# B&R Automation Studio project Panasonic_LinkaPowerCP2_A2021055 (part 27)

#### AtlasCopcoKomunikacia.st
```iecst
ACTION AtlasCopcoKomunikacia:

    M5_PrevodMomentu();
    K40_PrevodMomentu();

	//**************************************************************Skrutkovacka M5**************************************************************//
	//Vstupy z AtlasCopco do PLC//
    P3_Srobovanie.Skrutkovacka_M5.Stav_VysledokPotvrdeny:= P3_Srobovanie.PAR.M5_AtlasCopcoInputs[0].0;
    P3_Srobovanie.Skrutkovacka_M5.Stav_EmergencyStop:= P3_Srobovanie.PAR.M5_AtlasCopcoInputs[0].1;
    P3_Srobovanie.Skrutkovacka_M5.Stav_READY_to_START:= P3_Srobovanie.PAR.M5_AtlasCopcoInputs[0].2;
    P3_Srobovanie.Skrutkovacka_M5.Stav_MANUAL:= P3_Srobovanie.PAR.M5_AtlasCopcoInputs[0].3;
    P3_Srobovanie.Skrutkovacka_M5.Stav_UtahovanieUkoncene:= P3_Srobovanie.PAR.M5_AtlasCopcoInputs[0].4;
    P3_Srobovanie.Skrutkovacka_M5.Stav_VysledokUtahovania_NG:= P3_Srobovanie.PAR.M5_AtlasCopcoInputs[0].5;
    P3_Srobovanie.Skrutkovacka_M5.Stav_VysledokUtahovania_OK:= P3_Srobovanie.PAR.M5_AtlasCopcoInputs[0].6;
    P3_Srobovanie.Skrutkovacka_M5.Stav_SmerOtacania_VPRED:= P3_Srobovanie.PAR.M5_AtlasCopcoInputs[0].7;
    P3_Srobovanie.Skrutkovacka_M5.Stav_BUSY:= P3_Srobovanie.PAR.M5_AtlasCopcoInputs[0].8;
    P3_Srobovanie.Skrutkovacka_M5.Stav_ControlerSwitch_ON:= P3_Srobovanie.PAR.M5_AtlasCopcoInputs[0].9;
    P3_Srobovanie.Skrutkovacka_M5.Stav_Station_READY:= P3_Srobovanie.PAR.M5_AtlasCopcoInputs[0].10;
    P3_Srobovanie.Skrutkovacka_M5.Stav_NastrojPripojeny:= P3_Srobovanie.PAR.M5_AtlasCopcoInputs[0].11;
    P3_Srobovanie.Skrutkovacka_M5.Stav_NastrojUtahuje:= P3_Srobovanie.PAR.M5_AtlasCopcoInputs[0].12;

    //Výstupy z PLC do AtlasCopco//
    P3_Srobovanie.PAR.M5_AtlasCopcoOutputs[0].0:= P3_Srobovanie.Skrutkovacka_M5.RESET_Poruchy;
    P3_Srobovanie.PAR.M5_AtlasCopcoOutputs[0].1:= P3_Srobovanie.Skrutkovacka_M5.RESET_Vysledkov;
    P3_Srobovanie.PAR.M5_AtlasCopcoOutputs[0].2:= P3_Srobovanie.Skrutkovacka_M5.START_Skrutkovania;
    P3_Srobovanie.PAR.M5_AtlasCopcoOutputs[0].3:= P3_Srobovanie.Skrutkovacka_M5.START_Utahovania;

    //Dosiahnutý moment//
//    P3_Srobovanie.STAV.M5_DosiahnutyMoment.0:= P3_Srobovanie.PAR.M5_AtlasCopcoInputs[1].24;
//    P3_Srobovanie.STAV.M5_DosiahnutyMoment.1:= P3_Srobovanie.PAR.M5_AtlasCopcoInputs[1].25;
//    P3_Srobovanie.STAV.M5_DosiahnutyMoment.2:= P3_Srobovanie.PAR.M5_AtlasCopcoInputs[1].26;
//    P3_Srobovanie.STAV.M5_DosiahnutyMoment.3:= P3_Srobovanie.PAR.M5_AtlasCopcoInputs[1].27;
//    P3_Srobovanie.STAV.M5_DosiahnutyMoment.4:= P3_Srobovanie.PAR.M5_AtlasCopcoInputs[1].28;
//    P3_Srobovanie.STAV.M5_DosiahnutyMoment.5:= P3_Srobovanie.PAR.M5_AtlasCopcoInputs[1].29;
//    P3_Srobovanie.STAV.M5_DosiahnutyMoment.6:= P3_Srobovanie.PAR.M5_AtlasCopcoInputs[1].30;
//    P3_Srobovanie.STAV.M5_DosiahnutyMoment.7:= P3_Srobovanie.PAR.M5_AtlasCopcoInputs[1].31;
//    P3_Srobovanie.STAV.M5_DosiahnutyMoment.8:= P3_Srobovanie.PAR.M5_AtlasCopcoInputs[1].16;
//    P3_Srobovanie.STAV.M5_DosiahnutyMoment.9:= P3_Srobovanie.PAR.M5_AtlasCopcoInputs[1].17;
//    P3_Srobovanie.STAV.M5_DosiahnutyMoment.10:= P3_Srobovanie.PAR.M5_AtlasCopcoInputs[1].18;
//    P3_Srobovanie.STAV.M5_DosiahnutyMoment.11:= P3_Srobovanie.PAR.M5_AtlasCopcoInputs[1].19;
//    P3_Srobovanie.STAV.M5_DosiahnutyMoment.12:= P3_Srobovanie.PAR.M5_AtlasCopcoInputs[1].20;
//    P3_Srobovanie.STAV.M5_DosiahnutyMoment.13:= P3_Srobovanie.PAR.M5_AtlasCopcoInputs[1].21;
//    P3_Srobovanie.STAV.M5_DosiahnutyMoment.14:= P3_Srobovanie.PAR.M5_AtlasCopcoInputs[1].22;
//    P3_Srobovanie.STAV.M5_DosiahnutyMoment.15:= P3_Srobovanie.PAR.M5_AtlasCopcoInputs[1].23;
//    P3_Srobovanie.STAV.M5_DosiahnutyMoment.16:= P3_Srobovanie.PAR.M5_AtlasCopcoInputs[1].8;
//    P3_Srobovanie.STAV.M5_DosiahnutyMoment.17:= P3_Srobovanie.PAR.M5_AtlasCopcoInputs[1].9;
//    P3_Srobovanie.STAV.M5_DosiahnutyMoment.18:= P3_Srobovanie.PAR.M5_AtlasCopcoInputs[1].10;
//    P3_Srobovanie.STAV.M5_DosiahnutyMoment.19:= P3_Srobovanie.PAR.M5_AtlasCopcoInputs[1].11;
//    P3_Srobovanie.STAV.M5_DosiahnutyMoment.20:= P3_Srobovanie.PAR.M5_AtlasCopcoInputs[1].12;
//    P3_Srobovanie.STAV.M5_DosiahnutyMoment.21:= P3_Srobovanie.PAR.M5_AtlasCopcoInputs[1].13;
//    P3_Srobovanie.STAV.M5_DosiahnutyMoment.22:= P3_Srobovanie.PAR.M5_AtlasCopcoInputs[1].14;
//    P3_Srobovanie.STAV.M5_DosiahnutyMoment.23:= P3_Srobovanie.PAR.M5_AtlasCopcoInputs[1].15;
//    P3_Srobovanie.STAV.M5_DosiahnutyMoment.24:= P3_Srobovanie.PAR.M5_AtlasCopcoInputs[1].0;
//    P3_Srobovanie.STAV.M5_DosiahnutyMoment.25:= P3_Srobovanie.PAR.M5_AtlasCopcoInputs[1].1;
//    P3_Srobovanie.STAV.M5_DosiahnutyMoment.26:= P3_Srobovanie.PAR.M5_AtlasCopcoInputs[1].2;
//    P3_Srobovanie.STAV.M5_DosiahnutyMoment.27:= P3_Srobovanie.PAR.M5_AtlasCopcoInputs[1].3;
//    P3_Srobovanie.STAV.M5_DosiahnutyMoment.28:= P3_Srobovanie.PAR.M5_AtlasCopcoInputs[1].4;
//    P3_Srobovanie.STAV.M5_DosiahnutyMoment.29:= P3_Srobovanie.PAR.M5_AtlasCopcoInputs[1].5;
//    P3_Srobovanie.STAV.M5_DosiahnutyMoment.30:= P3_Srobovanie.PAR.M5_AtlasCopcoInputs[1].6;
//    P3_Srobovanie.STAV.M5_DosiahnutyMoment.31:= P3_Srobovanie.PAR.M5_AtlasCopcoInputs[1].7;
//    M5_DosiahnutyMoment_REAL:= UDINT_TO_REAL(P3_Srobovanie.STAV.M5_DosiahnutyMoment);
//    IF M5_DosiahnutyMoment_REAL > 0 THEN
//       P3_Srobovanie.STAV.M5_DosiahnutyMoment_REAL:= (M5_DosiahnutyMoment_REAL*2.34)/131106;
//    ELSE
//        P3_Srobovanie.STAV.M5_DosiahnutyMoment_REAL:= 0.0;
//    END_IF

    M5_PrevodMomentu.AtlasAktualnyMoment:=P3_Srobovanie.PAR.M5_AtlasCopcoInputs[1];
    P3_Srobovanie.STAV.M5_DosiahnutyMoment_REAL:=M5_PrevodMomentu.AktualnyMoment;

    (*P3_Srobovanie.STAV.M5_DosiahnutyMoment_REAL:= M5_DosiahnutyMoment_REAL /100;*)

    //Moment - Tolerancia MAX//
//    P3_Srobovanie.STAV.M5_Moment_ToleranciaMAX.0:= P3_Srobovanie.PAR.M5_AtlasCopcoInputs[3].24;
//    P3_Srobovanie.STAV.M5_Moment_ToleranciaMAX.1:= P3_Srobovanie.PAR.M5_AtlasCopcoInputs[3].25;
//    P3_Srobovanie.STAV.M5_Moment_ToleranciaMAX.2:= P3_Srobovanie.PAR.M5_AtlasCopcoInputs[3].26;
//    P3_Srobovanie.STAV.M5_Moment_ToleranciaMAX.3:= P3_Srobovanie.PAR.M5_AtlasCopcoInputs[3].27;
//    P3_Srobovanie.STAV.M5_Moment_ToleranciaMAX.4:= P3_Srobovanie.PAR.M5_AtlasCopcoInputs[3].28;
//    P3_Srobovanie.STAV.M5_Moment_ToleranciaMAX.5:= P3_Srobovanie.PAR.M5_AtlasCopcoInputs[3].29;
//    P3_Srobovanie.STAV.M5_Moment_ToleranciaMAX.6:= P3_Srobovanie.PAR.M5_AtlasCopcoInputs[3].30;
//    P3_Srobovanie.STAV.M5_Moment_ToleranciaMAX.7:= P3_Srobovanie.PAR.M5_AtlasCopcoInputs[3].31;
//    P3_Srobovanie.STAV.M5_Moment_ToleranciaMAX.8:= P3_Srobovanie.PAR.M5_AtlasCopcoInputs[3].16;
//    P3_Srobovanie.STAV.M5_Moment_ToleranciaMAX.9:= P3_Srobovanie.PAR.M5_AtlasCopcoInputs[3].17;
//    P3_Srobovanie.STAV.M5_Moment_ToleranciaMAX.10:= P3_Srobovanie.PAR.M5_AtlasCopcoInputs[3].18;
//    P3_Srobovanie.STAV.M5_Moment_ToleranciaMAX.11:= P3_Srobovanie.PAR.M5_AtlasCopcoInputs[3].19;
//    P3_Srobovanie.STAV.M5_Moment_ToleranciaMAX.12:= P3_Srobovanie.PAR.M5_AtlasCopcoInputs[3].20;
//    P3_Srobovanie.STAV.M5_Moment_ToleranciaMAX.13:= P3_Srobovanie.PAR.M5_AtlasCopcoInputs[3].21;
//    P3_Srobovanie.STAV.M5_Moment_ToleranciaMAX.14:= P3_Srobovanie.PAR.M5_AtlasCopcoInputs[3].22;
//    P3_Srobovanie.STAV.M5_Moment_ToleranciaMAX.15:= P3_Srobovanie.PAR.M5_AtlasCopcoInputs[3].23;
//    P3_Srobovanie.STAV.M5_Moment_ToleranciaMAX.16:= P3_Srobovanie.PAR.M5_AtlasCopcoInputs[3].8;
//    P3_Srobovanie.STAV.M5_Moment_ToleranciaMAX.17:= P3_Srobovanie.PAR.M5_AtlasCopcoInputs[3].9;
//    P3_Srobovanie.STAV.M5_Moment_ToleranciaMAX.18:= P3_Srobovanie.PAR.M5_AtlasCopcoInputs[3].10;
//    P3_Srobovanie.STAV.M5_Moment_ToleranciaMAX.19:= P3_Srobovanie.PAR.M5_AtlasCopcoInputs[3].11;
//    P3_Srobovanie.STAV.M5_Moment_ToleranciaMAX.20:= P3_Srobovanie.PAR.M5_AtlasCopcoInputs[3].12;
//    P3_Srobovanie.STAV.M5_Moment_ToleranciaMAX.21:= P3_Srobovanie.PAR.M5_AtlasCopcoInputs[3].13;
//    P3_Srobovanie.STAV.M5_Moment_ToleranciaMAX.22:= P3_Srobovanie.PAR.M5_AtlasCopcoInputs[3].14;
//    P3_Srobovanie.STAV.M5_Moment_ToleranciaMAX.23:= P3_Srobovanie.PAR.M5_AtlasCopcoInputs[3].15;
//    P3_Srobovanie.STAV.M5_Moment_ToleranciaMAX.24:= P3_Srobovanie.PAR.M5_AtlasCopcoInputs[3].0;
//    P3_Srobovanie.STAV.M5_Moment_ToleranciaMAX.25:= P3_Srobovanie.PAR.M5_AtlasCopcoInputs[3].1;
//    P3_Srobovanie.STAV.M5_Moment_ToleranciaMAX.26:= P3_Srobovanie.PAR.M5_AtlasCopcoInputs[3].2;
//    P3_Srobovanie.STAV.M5_Moment_ToleranciaMAX.27:= P3_Srobovanie.PAR.M5_AtlasCopcoInputs[3].3;
//    P3_Srobovanie.STAV.M5_Moment_ToleranciaMAX.28:= P3_Srobovanie.PAR.M5_AtlasCopcoInputs[3].4;
//    P3_Srobovanie.STAV.M5_Moment_ToleranciaMAX.29:= P3_Srobovanie.PAR.M5_AtlasCopcoInputs[3].5;
//    P3_Srobovanie.STAV.M5_Moment_ToleranciaMAX.30:= P3_Srobovanie.PAR.M5_AtlasCopcoInputs[3].6;
//    P3_Srobovanie.STAV.M5_Moment_ToleranciaMAX.31:= P3_Srobovanie.PAR.M5_AtlasCopcoInputs[3].7;
//    M5_Moment_ToleranciaMAX_REAL:= UDINT_TO_REAL(P3_Srobovanie.STAV.M5_Moment_ToleranciaMAX);
//    IF M5_Moment_ToleranciaMAX_REAL > 0 THEN
//      P3_Srobovanie.STAV.M5_Moment_ToleranciaMAX_REAL:= (M5_Moment_ToleranciaMAX_REAL*2.82)/131154;
//    ELSE
//        P3_Srobovanie.STAV.M5_Moment_ToleranciaMAX_REAL:= 0.0;
//    END_IF
//

    M5_PrevodMomentu.AtlasMaximalnaTolerancia:=P3_Srobovanie.PAR.M5_AtlasCopcoInputs[3];
    P3_Srobovanie.STAV.M5_Moment_ToleranciaMAX_REAL:=M5_PrevodMomentu.ToleranciaMAX;

    (*P3_Srobovanie.STAV.M5_Moment_ToleranciaMAX_REAL:= M5_Moment_ToleranciaMAX_REAL /100;*)

    //Moment - Tolerancia MIN//
//    P3_Srobovanie.STAV.M5_Moment_ToleranciaMIN.0:= P3_Srobovanie.PAR.M5_AtlasCopcoInputs[4].24;
//    P3_Srobovanie.STAV.M5_Moment_ToleranciaMIN.1:= P3_Srobovanie.PAR.M5_AtlasCopcoInputs[4].25;
//    P3_Srobovanie.STAV.M5_Moment_ToleranciaMIN.2:= P3_Srobovanie.PAR.M5_AtlasCopcoInputs[4].26;
//    P3_Srobovanie.STAV.M5_Moment_ToleranciaMIN.3:= P3_Srobovanie.PAR.M5_AtlasCopcoInputs[4].27;
//    P3_Srobovanie.STAV.M5_Moment_ToleranciaMIN.4:= P3_Srobovanie.PAR.M5_AtlasCopcoInputs[4].28;
//    P3_Srobovanie.STAV.M5_Moment_ToleranciaMIN.5:= P3_Srobovanie.PAR.M5_AtlasCopcoInputs[4].29;
//    P3_Srobovanie.STAV.M5_Moment_ToleranciaMIN.6:= P3_Srobovanie.PAR.M5_AtlasCopcoInputs[4].30;
//    P3_Srobovanie.STAV.M5_Moment_ToleranciaMIN.7:= P3_Srobovanie.PAR.M5_AtlasCopcoInputs[4].31;
//    P3_Srobovanie.STAV.M5_Moment_ToleranciaMIN.8:= P3_Srobovanie.PAR.M5_AtlasCopcoInputs[4].16;
//    P3_Srobovanie.STAV.M5_Moment_ToleranciaMIN.9:= P3_Srobovanie.PAR.M5_AtlasCopcoInputs[4].17;
//    P3_Srobovanie.STAV.M5_Moment_ToleranciaMIN.10:= P3_Srobovanie.PAR.M5_AtlasCopcoInputs[4].18;
//    P3_Srobovanie.STAV.M5_Moment_ToleranciaMIN.11:= P3_Srobovanie.PAR.M5_AtlasCopcoInputs[4].19;
//    P3_Srobovanie.STAV.M5_Moment_ToleranciaMIN.12:= P3_Srobovanie.PAR.M5_AtlasCopcoInputs[4].20;
//    P3_Srobovanie.STAV.M5_Moment_ToleranciaMIN.13:= P3_Srobovanie.PAR.M5_AtlasCopcoInputs[4].21;
//    P3_Srobovanie.STAV.M5_Moment_ToleranciaMIN.14:= P3_Srobovanie.PAR.M5_AtlasCopcoInputs[4].22;
//    P3_Srobovanie.STAV.M5_Moment_ToleranciaMIN.15:= P3_Srobovanie.PAR.M5_AtlasCopcoInputs[4].23;
//    P3_Srobovanie.STAV.M5_Moment_ToleranciaMIN.16:= P3_Srobovanie.PAR.M5_AtlasCopcoInputs[4].8;
//    P3_Srobovanie.STAV.M5_Moment_ToleranciaMIN.17:= P3_Srobovanie.PAR.M5_AtlasCopcoInputs[4].9;
//    P3_Srobovanie.STAV.M5_Moment_ToleranciaMIN.18:= P3_Srobovanie.PAR.M5_AtlasCopcoInputs[4].10;
//    P3_Srobovanie.STAV.M5_Moment_ToleranciaMIN.19:= P3_Srobovanie.PAR.M5_AtlasCopcoInputs[4].11;
//    P3_Srobovanie.STAV.M5_Moment_ToleranciaMIN.20:= P3_Srobovanie.PAR.M5_AtlasCopcoInputs[4].12;
//    P3_Srobovanie.STAV.M5_Moment_ToleranciaMIN.21:= P3_Srobovanie.PAR.M5_AtlasCopcoInputs[4].13;
//    P3_Srobovanie.STAV.M5_Moment_ToleranciaMIN.22:= P3_Srobovanie.PAR.M5_AtlasCopcoInputs[4].14;
//    P3_Srobovanie.STAV.M5_Moment_ToleranciaMIN.23:= P3_Srobovanie.PAR.M5_AtlasCopcoInputs[4].15;
//    P3_Srobovanie.STAV.M5_Moment_ToleranciaMIN.24:= P3_Srobovanie.PAR.M5_AtlasCopcoInputs[4].0;
//    P3_Srobovanie.STAV.M5_Moment_ToleranciaMIN.25:= P3_Srobovanie.PAR.M5_AtlasCopcoInputs[4].1;
//    P3_Srobovanie.STAV.M5_Moment_ToleranciaMIN.26:= P3_Srobovanie.PAR.M5_AtlasCopcoInputs[4].2;
//    P3_Srobovanie.STAV.M5_Moment_ToleranciaMIN.27:= P3_Srobovanie.PAR.M5_AtlasCopcoInputs[4].3;
//    P3_Srobovanie.STAV.M5_Moment_ToleranciaMIN.28:= P3_Srobovanie.PAR.M5_AtlasCopcoInputs[4].4;
//    P3_Srobovanie.STAV.M5_Moment_ToleranciaMIN.29:= P3_Srobovanie.PAR.M5_AtlasCopcoInputs[4].5;
//    P3_Srobovanie.STAV.M5_Moment_ToleranciaMIN.30:= P3_Srobovanie.PAR.M5_AtlasCopcoInputs[4].6;
//    P3_Srobovanie.STAV.M5_Moment_ToleranciaMIN.31:= P3_Srobovanie.PAR.M5_AtlasCopcoInputs[4].7;
//    M5_Moment_ToleranciaMIN_REAL:= UDINT_TO_REAL(P3_Srobovanie.STAV.M5_Moment_ToleranciaMIN);
//    IF M5_Moment_ToleranciaMIN_REAL > 0 THEN
//       P3_Srobovanie.STAV.M5_Moment_ToleranciaMIN_REAL:= (M5_Moment_ToleranciaMIN_REAL*2.34)/131106;
//    ELSE
//        P3_Srobovanie.STAV.M5_Moment_ToleranciaMIN_REAL:= 0.0;
//    END_IF

    M5_PrevodMomentu.AtlasMinimalnaTolerancia:=P3_Srobovanie.PAR.M5_AtlasCopcoInputs[4];
    P3_Srobovanie.STAV.M5_Moment_ToleranciaMIN_REAL:=M5_PrevodMomentu.ToleranciaMIN;

    (*P3_Srobovanie.STAV.M5_Moment_ToleranciaMIN_REAL:= M5_Moment_ToleranciaMIN_REAL/100;*)

    //Dosiahnutý úhol//
    P3_Srobovanie.STAV.M5_DosiahnutyUhol.0:= P3_Srobovanie.PAR.M5_AtlasCopcoInputs[0].24;
    P3_Srobovanie.STAV.M5_DosiahnutyUhol.1:= P3_Srobovanie.PAR.M5_AtlasCopcoInputs[0].25;
    P3_Srobovanie.STAV.M5_DosiahnutyUhol.2:= P3_Srobovanie.PAR.M5_AtlasCopcoInputs[0].26;
    P3_Srobovanie.STAV.M5_DosiahnutyUhol.3:= P3_Srobovanie.PAR.M5_AtlasCopcoInputs[0].27;
    P3_Srobovanie.STAV.M5_DosiahnutyUhol.4:= P3_Srobovanie.PAR.M5_AtlasCopcoInputs[0].28;
    P3_Srobovanie.STAV.M5_DosiahnutyUhol.5:= P3_Srobovanie.PAR.M5_AtlasCopcoInputs[0].29;
    P3_Srobovanie.STAV.M5_DosiahnutyUhol.6:= P3_Srobovanie.PAR.M5_AtlasCopcoInputs[0].30;
    P3_Srobovanie.STAV.M5_DosiahnutyUhol.7:= P3_Srobovanie.PAR.M5_AtlasCopcoInputs[0].31;
    P3_Srobovanie.STAV.M5_DosiahnutyUhol.8:= P3_Srobovanie.PAR.M5_AtlasCopcoInputs[0].16;
    P3_Srobovanie.STAV.M5_DosiahnutyUhol.9:= P3_Srobovanie.PAR.M5_AtlasCopcoInputs[0].17;
    P3_Srobovanie.STAV.M5_DosiahnutyUhol.10:= P3_Srobovanie.PAR.M5_AtlasCopcoInputs[0].18;
    P3_Srobovanie.STAV.M5_DosiahnutyUhol.11:= P3_Srobovanie.PAR.M5_AtlasCopcoInputs[0].19;
    P3_Srobovanie.STAV.M5_DosiahnutyUhol.12:= P3_Srobovanie.PAR.M5_AtlasCopcoInputs[0].20;
    P3_Srobovanie.STAV.M5_DosiahnutyUhol.13:= P3_Srobovanie.PAR.M5_AtlasCopcoInputs[0].21;
    P3_Srobovanie.STAV.M5_DosiahnutyUhol.14:= P3_Srobovanie.PAR.M5_AtlasCopcoInputs[0].22;
    P3_Srobovanie.STAV.M5_DosiahnutyUhol.15:= P3_Srobovanie.PAR.M5_AtlasCopcoInputs[0].23;

    //Uhol - Tolerancia MAX//
    P3_Srobovanie.STAV.M5_Uhol_ToleranciaMAX.0:= P3_Srobovanie.PAR.M5_AtlasCopcoInputs[2].8;
    P3_Srobovanie.STAV.M5_Uhol_ToleranciaMAX.1:= P3_Srobovanie.PAR.M5_AtlasCopcoInputs[2].9;
    P3_Srobovanie.STAV.M5_Uhol_ToleranciaMAX.2:= P3_Srobovanie.PAR.M5_AtlasCopcoInputs[2].10;
    P3_Srobovanie.STAV.M5_Uhol_ToleranciaMAX.3:= P3_Srobovanie.PAR.M5_AtlasCopcoInputs[2].11;
    P3_Srobovanie.STAV.M5_Uhol_ToleranciaMAX.4:= P3_Srobovanie.PAR.M5_AtlasCopcoInputs[2].12;
    P3_Srobovanie.STAV.M5_Uhol_ToleranciaMAX.5:= P3_Srobovanie.PAR.M5_AtlasCopcoInputs[2].13;
    P3_Srobovanie.STAV.M5_Uhol_ToleranciaMAX.6:= P3_Srobovanie.PAR.M5_AtlasCopcoInputs[2].14;
    P3_Srobovanie.STAV.M5_Uhol_ToleranciaMAX.7:= P3_Srobovanie.PAR.M5_AtlasCopcoInputs[2].15;
    P3_Srobovanie.STAV.M5_Uhol_ToleranciaMAX.8:= P3_Srobovanie.PAR.M5_AtlasCopcoInputs[2].0;
    P3_Srobovanie.STAV.M5_Uhol_ToleranciaMAX.9:= P3_Srobovanie.PAR.M5_AtlasCopcoInputs[2].1;
    P3_Srobovanie.STAV.M5_Uhol_ToleranciaMAX.10:= P3_Srobovanie.PAR.M5_AtlasCopcoInputs[2].2;
    P3_Srobovanie.STAV.M5_Uhol_ToleranciaMAX.11:= P3_Srobovanie.PAR.M5_AtlasCopcoInputs[2].3;
    P3_Srobovanie.STAV.M5_Uhol_ToleranciaMAX.12:= P3_Srobovanie.PAR.M5_AtlasCopcoInputs[2].4;
    P3_Srobovanie.STAV.M5_Uhol_ToleranciaMAX.13:= P3_Srobovanie.PAR.M5_AtlasCopcoInputs[2].5;
    P3_Srobovanie.STAV.M5_Uhol_ToleranciaMAX.14:= P3_Srobovanie.PAR.M5_AtlasCopcoInputs[2].6;
    P3_Srobovanie.STAV.M5_Uhol_ToleranciaMAX.15:= P3_Srobovanie.PAR.M5_AtlasCopcoInputs[2].7;

    //Uhol - Tolerancia MIN//
    P3_Srobovanie.STAV.M5_Uhol_ToleranciaMIN.0:= P3_Srobovanie.PAR.M5_AtlasCopcoInputs[2].24;
    P3_Srobovanie.STAV.M5_Uhol_ToleranciaMIN.1:= P3_Srobovanie.PAR.M5_AtlasCopcoInputs[2].25;
    P3_Srobovanie.STAV.M5_Uhol_ToleranciaMIN.2:= P3_Srobovanie.PAR.M5_AtlasCopcoInputs[2].26;
    P3_Srobovanie.STAV.M5_Uhol_ToleranciaMIN.3:= P3_Srobovanie.PAR.M5_AtlasCopcoInputs[2].27;
    P3_Srobovanie.STAV.M5_Uhol_ToleranciaMIN.4:= P3_Srobovanie.PAR.M5_AtlasCopcoInputs[2].28;
    P3_Srobovanie.STAV.M5_Uhol_ToleranciaMIN.5:= P3_Srobovanie.PAR.M5_AtlasCopcoInputs[2].29;
    P3_Srobovanie.STAV.M5_Uhol_ToleranciaMIN.6:= P3_Srobovanie.PAR.M5_AtlasCopcoInputs[2].30;
    P3_Srobovanie.STAV.M5_Uhol_ToleranciaMIN.7:= P3_Srobovanie.PAR.M5_AtlasCopcoInputs[2].31;
    P3_Srobovanie.STAV.M5_Uhol_ToleranciaMIN.8:= P3_Srobovanie.PAR.M5_AtlasCopcoInputs[2].16;
    P3_Srobovanie.STAV.M5_Uhol_ToleranciaMIN.9:= P3_Srobovanie.PAR.M5_AtlasCopcoInputs[2].17;
    P3_Srobovanie.STAV.M5_Uhol_ToleranciaMIN.10:= P3_Srobovanie.PAR.M5_AtlasCopcoInputs[2].18;
    P3_Srobovanie.STAV.M5_Uhol_ToleranciaMIN.11:= P3_Srobovanie.PAR.M5_AtlasCopcoInputs[2].19;
    P3_Srobovanie.STAV.M5_Uhol_ToleranciaMIN.12:= P3_Srobovanie.PAR.M5_AtlasCopcoInputs[2].20;
    P3_Srobovanie.STAV.M5_Uhol_ToleranciaMIN.13:= P3_Srobovanie.PAR.M5_AtlasCopcoInputs[2].21;
    P3_Srobovanie.STAV.M5_Uhol_ToleranciaMIN.14:= P3_Srobovanie.PAR.M5_AtlasCopcoInputs[2].22;
    P3_Srobovanie.STAV.M5_Uhol_ToleranciaMIN.15:= P3_Srobovanie.PAR.M5_AtlasCopcoInputs[2].23;

    //***********************************************Skrutkovacka K40**********************************************************************//
    //Vstupy z AtlasCopco do PLC//
    P3_Srobovanie.Skrutkovacka_K40.Stav_VysledokPotvrdeny:= P3_Srobovanie.PAR.K40_AtlasCopcoInputs[0].0;
    P3_Srobovanie.Skrutkovacka_K40.Stav_EmergencyStop:= P3_Srobovanie.PAR.K40_AtlasCopcoInputs[0].1;
    P3_Srobovanie.Skrutkovacka_K40.Stav_READY_to_START:= P3_Srobovanie.PAR.K40_AtlasCopcoInputs[0].2;
    P3_Srobovanie.Skrutkovacka_K40.Stav_MANUAL:= P3_Srobovanie.PAR.K40_AtlasCopcoInputs[0].3;
    P3_Srobovanie.Skrutkovacka_K40.Stav_UtahovanieUkoncene:= P3_Srobovanie.PAR.K40_AtlasCopcoInputs[0].4;
    P3_Srobovanie.Skrutkovacka_K40.Stav_VysledokUtahovania_NG:= P3_Srobovanie.PAR.K40_AtlasCopcoInputs[0].5;
    P3_Srobovanie.Skrutkovacka_K40.Stav_VysledokUtahovania_OK:= P3_Srobovanie.PAR.K40_AtlasCopcoInputs[0].6;
    P3_Srobovanie.Skrutkovacka_K40.Stav_SmerOtacania_VPRED:= P3_Srobovanie.PAR.K40_AtlasCopcoInputs[0].7;
    P3_Srobovanie.Skrutkovacka_K40.Stav_BUSY:= P3_Srobovanie.PAR.K40_AtlasCopcoInputs[0].8;
    P3_Srobovanie.Skrutkovacka_K40.Stav_ControlerSwitch_ON:= P3_Srobovanie.PAR.K40_AtlasCopcoInputs[0].9;
    P3_Srobovanie.Skrutkovacka_K40.Stav_Station_READY:= P3_Srobovanie.PAR.K40_AtlasCopcoInputs[0].10;
    P3_Srobovanie.Skrutkovacka_K40.Stav_NastrojPripojeny:= P3_Srobovanie.PAR.K40_AtlasCopcoInputs[0].11;
    P3_Srobovanie.Skrutkovacka_K40.Stav_NastrojUtahuje:= P3_Srobovanie.PAR.K40_AtlasCopcoInputs[0].12;

    //Výstupy z PLC do AtlasCopco//
    P3_Srobovanie.PAR.K40_AtlasCopcoOutputs[0].0:= P3_Srobovanie.Skrutkovacka_K40.RESET_Poruchy;
    P3_Srobovanie.PAR.K40_AtlasCopcoOutputs[0].1:= P3_Srobovanie.Skrutkovacka_K40.RESET_Vysledkov;
    P3_Srobovanie.PAR.K40_AtlasCopcoOutputs[0].2:= P3_Srobovanie.Skrutkovacka_K40.START_Skrutkovania;
    P3_Srobovanie.PAR.K40_AtlasCopcoOutputs[0].3:= P3_Srobovanie.Skrutkovacka_K40.START_Utahovania;

    //Dosiahnutý moment//
//    P3_Srobovanie.STAV.K40_DosiahnutyMoment.0:= P3_Srobovanie.PAR.K40_AtlasCopcoInputs[1].24;
//    P3_Srobovanie.STAV.K40_DosiahnutyMoment.1:= P3_Srobovanie.PAR.K40_AtlasCopcoInputs[1].25;
//    P3_Srobovanie.STAV.K40_DosiahnutyMoment.2:= P3_Srobovanie.PAR.K40_AtlasCopcoInputs[1].26;
//    P3_Srobovanie.STAV.K40_DosiahnutyMoment.3:= P3_Srobovanie.PAR.K40_AtlasCopcoInputs[1].27;
//    P3_Srobovanie.STAV.K40_DosiahnutyMoment.4:= P3_Srobovanie.PAR.K40_AtlasCopcoInputs[1].28;
//    P3_Srobovanie.STAV.K40_DosiahnutyMoment.5:= P3_Srobovanie.PAR.K40_AtlasCopcoInputs[1].29;
//    P3_Srobovanie.STAV.K40_DosiahnutyMoment.6:= P3_Srobovanie.PAR.K40_AtlasCopcoInputs[1].30;
//    P3_Srobovanie.STAV.K40_DosiahnutyMoment.7:= P3_Srobovanie.PAR.K40_AtlasCopcoInputs[1].31;
//    P3_Srobovanie.STAV.K40_DosiahnutyMoment.8:= P3_Srobovanie.PAR.K40_AtlasCopcoInputs[1].16;
//    P3_Srobovanie.STAV.K40_DosiahnutyMoment.9:= P3_Srobovanie.PAR.K40_AtlasCopcoInputs[1].17;
//    P3_Srobovanie.STAV.K40_DosiahnutyMoment.10:= P3_Srobovanie.PAR.K40_AtlasCopcoInputs[1].18;
//    P3_Srobovanie.STAV.K40_DosiahnutyMoment.11:= P3_Srobovanie.PAR.K40_AtlasCopcoInputs[1].19;
//    P3_Srobovanie.STAV.K40_DosiahnutyMoment.12:= P3_Srobovanie.PAR.K40_AtlasCopcoInputs[1].20;
//    P3_Srobovanie.STAV.K40_DosiahnutyMoment.13:= P3_Srobovanie.PAR.K40_AtlasCopcoInputs[1].21;
//    P3_Srobovanie.STAV.K40_DosiahnutyMoment.14:= P3_Srobovanie.PAR.K40_AtlasCopcoInputs[1].22;
//    P3_Srobovanie.STAV.K40_DosiahnutyMoment.15:= P3_Srobovanie.PAR.K40_AtlasCopcoInputs[1].23;
//    P3_Srobovanie.STAV.K40_DosiahnutyMoment.16:= P3_Srobovanie.PAR.K40_AtlasCopcoInputs[1].8;
//    P3_Srobovanie.STAV.K40_DosiahnutyMoment.17:= P3_Srobovanie.PAR.K40_AtlasCopcoInputs[1].9;
//    P3_Srobovanie.STAV.K40_DosiahnutyMoment.18:= P3_Srobovanie.PAR.K40_AtlasCopcoInputs[1].10;
//    P3_Srobovanie.STAV.K40_DosiahnutyMoment.19:= P3_Srobovanie.PAR.K40_AtlasCopcoInputs[1].11;
//    P3_Srobovanie.STAV.K40_DosiahnutyMoment.20:= P3_Srobovanie.PAR.K40_AtlasCopcoInputs[1].12;
//    P3_Srobovanie.STAV.K40_DosiahnutyMoment.21:= P3_Srobovanie.PAR.K40_AtlasCopcoInputs[1].13;
//    P3_Srobovanie.STAV.K40_DosiahnutyMoment.22:= P3_Srobovanie.PAR.K40_AtlasCopcoInputs[1].14;
//    P3_Srobovanie.STAV.K40_DosiahnutyMoment.23:= P3_Srobovanie.PAR.K40_AtlasCopcoInputs[1].15;
//    P3_Srobovanie.STAV.K40_DosiahnutyMoment.24:= P3_Srobovanie.PAR.K40_AtlasCopcoInputs[1].0;
//    P3_Srobovanie.STAV.K40_DosiahnutyMoment.25:= P3_Srobovanie.PAR.K40_AtlasCopcoInputs[1].1;
//    P3_Srobovanie.STAV.K40_DosiahnutyMoment.26:= P3_Srobovanie.PAR.K40_AtlasCopcoInputs[1].2;
//    P3_Srobovanie.STAV.K40_DosiahnutyMoment.27:= P3_Srobovanie.PAR.K40_AtlasCopcoInputs[1].3;
//    P3_Srobovanie.STAV.K40_DosiahnutyMoment.28:= P3_Srobovanie.PAR.K40_AtlasCopcoInputs[1].4;
//    P3_Srobovanie.STAV.K40_DosiahnutyMoment.29:= P3_Srobovanie.PAR.K40_AtlasCopcoInputs[1].5;
//    P3_Srobovanie.STAV.K40_DosiahnutyMoment.30:= P3_Srobovanie.PAR.K40_AtlasCopcoInputs[1].6;
//    P3_Srobovanie.STAV.K40_DosiahnutyMoment.31:= P3_Srobovanie.PAR.K40_AtlasCopcoInputs[1].7;
//    K40_DosiahnutyMoment_REAL:= UDINT_TO_REAL(P3_Srobovanie.STAV.K40_DosiahnutyMoment);
//    IF K40_DosiahnutyMoment_REAL > 0 THEN
//        P3_Srobovanie.STAV.K40_DosiahnutyMoment_REAL:= (K40_DosiahnutyMoment_REAL*1.35)/65571;
//    ELSE
//        P3_Srobovanie.STAV.K40_DosiahnutyMoment_REAL:=0.0;
//    END_IF

    K40_PrevodMomentu.AtlasAktualnyMoment:=P3_Srobovanie.PAR.K40_AtlasCopcoInputs[1];
    P3_Srobovanie.STAV.K40_DosiahnutyMoment_REAL:=K40_PrevodMomentu.AktualnyMoment;

    (*P3_Srobovanie.STAV.K40_DosiahnutyMoment_REAL:= K40_DosiahnutyMoment_REAL/100;*)

    //Moment - Tolerancia MAX//
//    P3_Srobovanie.STAV.K40_Moment_ToleranciaMAX.0:= P3_Srobovanie.PAR.K40_AtlasCopcoInputs[3].24;
//    P3_Srobovanie.STAV.K40_Moment_ToleranciaMAX.1:= P3_Srobovanie.PAR.K40_AtlasCopcoInputs[3].25;
//    P3_Srobovanie.STAV.K40_Moment_ToleranciaMAX.2:= P3_Srobovanie.PAR.K40_AtlasCopcoInputs[3].26;
//    P3_Srobovanie.STAV.K40_Moment_ToleranciaMAX.3:= P3_Srobovanie.PAR.K40_AtlasCopcoInputs[3].27;
//    P3_Srobovanie.STAV.K40_Moment_ToleranciaMAX.4:= P3_Srobovanie.PAR.K40_AtlasCopcoInputs[3].28;
//    P3_Srobovanie.STAV.K40_Moment_ToleranciaMAX.5:= P3_Srobovanie.PAR.K40_AtlasCopcoInputs[3].29;
//    P3_Srobovanie.STAV.K40_Moment_ToleranciaMAX.6:= P3_Srobovanie.PAR.K40_AtlasCopcoInputs[3].30;
//    P3_Srobovanie.STAV.K40_Moment_ToleranciaMAX.7:= P3_Srobovanie.PAR.K40_AtlasCopcoInputs[3].31;
//    P3_Srobovanie.STAV.K40_Moment_ToleranciaMAX.8:= P3_Srobovanie.PAR.K40_AtlasCopcoInputs[3].16;
//    P3_Srobovanie.STAV.K40_Moment_ToleranciaMAX.9:= P3_Srobovanie.PAR.K40_AtlasCopcoInputs[3].17;
//    P3_Srobovanie.STAV.K40_Moment_ToleranciaMAX.10:= P3_Srobovanie.PAR.K40_AtlasCopcoInputs[3].18;
//    P3_Srobovanie.STAV.K40_Moment_ToleranciaMAX.11:= P3_Srobovanie.PAR.K40_AtlasCopcoInputs[3].19;
//    P3_Srobovanie.STAV.K40_Moment_ToleranciaMAX.12:= P3_Srobovanie.PAR.K40_AtlasCopcoInputs[3].20;
//    P3_Srobovanie.STAV.K40_Moment_ToleranciaMAX.13:= P3_Srobovanie.PAR.K40_AtlasCopcoInputs[3].21;
//    P3_Srobovanie.STAV.K40_Moment_ToleranciaMAX.14:= P3_Srobovanie.PAR.K40_AtlasCopcoInputs[3].22;
//    P3_Srobovanie.STAV.K40_Moment_ToleranciaMAX.15:= P3_Srobovanie.PAR.K40_AtlasCopcoInputs[3].23;
//    P3_Srobovanie.STAV.K40_Moment_ToleranciaMAX.16:= P3_Srobovanie.PAR.K40_AtlasCopcoInputs[3].8;
//    P3_Srobovanie.STAV.K40_Moment_ToleranciaMAX.17:= P3_Srobovanie.PAR.K40_AtlasCopcoInputs[3].9;
//    P3_Srobovanie.STAV.K40_Moment_ToleranciaMAX.18:= P3_Srobovanie.PAR.K40_AtlasCopcoInputs[3].10;
//    P3_Srobovanie.STAV.K40_Moment_ToleranciaMAX.19:= P3_Srobovanie.PAR.K40_AtlasCopcoInputs[3].11;
//    P3_Srobovanie.STAV.K40_Moment_ToleranciaMAX.20:= P3_Srobovanie.PAR.K40_AtlasCopcoInputs[3].12;
//    P3_Srobovanie.STAV.K40_Moment_ToleranciaMAX.21:= P3_Srobovanie.PAR.K40_AtlasCopcoInputs[3].13;
//    P3_Srobovanie.STAV.K40_Moment_ToleranciaMAX.22:= P3_Srobovanie.PAR.K40_AtlasCopcoInputs[3].14;
//    P3_Srobovanie.STAV.K40_Moment_ToleranciaMAX.23:= P3_Srobovanie.PAR.K40_AtlasCopcoInputs[3].15;
//    P3_Srobovanie.STAV.K40_Moment_ToleranciaMAX.24:= P3_Srobovanie.PAR.K40_AtlasCopcoInputs[3].0;
//    P3_Srobovanie.STAV.K40_Moment_ToleranciaMAX.25:= P3_Srobovanie.PAR.K40_AtlasCopcoInputs[3].1;
//    P3_Srobovanie.STAV.K40_Moment_ToleranciaMAX.26:= P3_Srobovanie.PAR.K40_AtlasCopcoInputs[3].2;
//    P3_Srobovanie.STAV.K40_Moment_ToleranciaMAX.27:= P3_Srobovanie.PAR.K40_AtlasCopcoInputs[3].3;
//    P3_Srobovanie.STAV.K40_Moment_ToleranciaMAX.28:= P3_Srobovanie.PAR.K40_AtlasCopcoInputs[3].4;
//    P3_Srobovanie.STAV.K40_Moment_ToleranciaMAX.29:= P3_Srobovanie.PAR.K40_AtlasCopcoInputs[3].5;
//    P3_Srobovanie.STAV.K40_Moment_ToleranciaMAX.30:= P3_Srobovanie.PAR.K40_AtlasCopcoInputs[3].6;
//    P3_Srobovanie.STAV.K40_Moment_ToleranciaMAX.31:= P3_Srobovanie.PAR.K40_AtlasCopcoInputs[3].7;
//    K40_Moment_ToleranciaMAX_REAL:= UDINT_TO_REAL(P3_Srobovanie.STAV.K40_Moment_ToleranciaMAX);
//    IF K40_Moment_ToleranciaMAX_REAL > 0 THEN
//       P3_Srobovanie.STAV.K40_Moment_ToleranciaMAX_REAL:= (K40_Moment_ToleranciaMAX_REAL*1.65)/65601;
//    ELSE
//        P3_Srobovanie.STAV.K40_Moment_ToleranciaMAX_REAL:= 0.0;
//    END_IF

    K40_PrevodMomentu.AtlasMaximalnaTolerancia:=P3_Srobovanie.PAR.K40_AtlasCopcoInputs[3];
    P3_Srobovanie.STAV.K40_Moment_ToleranciaMAX_REAL:=K40_PrevodMomentu.ToleranciaMAX;

    (*P3_Srobovanie.STAV.K40_Moment_ToleranciaMAX_REAL:= K40_Moment_ToleranciaMAX_REAL/100;*)

    //Moment - Tolerancia MIN//
//    P3_Srobovanie.STAV.K40_Moment_ToleranciaMIN.0:= P3_Srobovanie.PAR.K40_AtlasCopcoInputs[4].24;
//    P3_Srobovanie.STAV.K40_Moment_ToleranciaMIN.1:= P3_Srobovanie.PAR.K40_AtlasCopcoInputs[4].25;
//    P3_Srobovanie.STAV.K40_Moment_ToleranciaMIN.2:= P3_Srobovanie.PAR.K40_AtlasCopcoInputs[4].26;
//    P3_Srobovanie.STAV.K40_Moment_ToleranciaMIN.3:= P3_Srobovanie.PAR.K40_AtlasCopcoInputs[4].27;
//    P3_Srobovanie.STAV.K40_Moment_ToleranciaMIN.4:= P3_Srobovanie.PAR.K40_AtlasCopcoInputs[4].28;
//    P3_Srobovanie.STAV.K40_Moment_ToleranciaMIN.5:= P3_Srobovanie.PAR.K40_AtlasCopcoInputs[4].29;
//    P3_Srobovanie.STAV.K40_Moment_ToleranciaMIN.6:= P3_Srobovanie.PAR.K40_AtlasCopcoInputs[4].30;
//    P3_Srobovanie.STAV.K40_Moment_ToleranciaMIN.7:= P3_Srobovanie.PAR.K40_AtlasCopcoInputs[4].31;
//    P3_Srobovanie.STAV.K40_Moment_ToleranciaMIN.8:= P3_Srobovanie.PAR.K40_AtlasCopcoInputs[4].16;
//    P3_Srobovanie.STAV.K40_Moment_ToleranciaMIN.9:= P3_Srobovanie.PAR.K40_AtlasCopcoInputs[4].17;
//    P3_Srobovanie.STAV.K40_Moment_ToleranciaMIN.10:= P3_Srobovanie.PAR.K40_AtlasCopcoInputs[4].18;
//    P3_Srobovanie.STAV.K40_Moment_ToleranciaMIN.11:= P3_Srobovanie.PAR.K40_AtlasCopcoInputs[4].19;
//    P3_Srobovanie.STAV.K40_Moment_ToleranciaMIN.12:= P3_Srobovanie.PAR.K40_AtlasCopcoInputs[4].20;
//    P3_Srobovanie.STAV.K40_Moment_ToleranciaMIN.13:= P3_Srobovanie.PAR.K40_AtlasCopcoInputs[4].21;
//    P3_Srobovanie.STAV.K40_Moment_ToleranciaMIN.14:= P3_Srobovanie.PAR.K40_AtlasCopcoInputs[4].22;
//    P3_Srobovanie.STAV.K40_Moment_ToleranciaMIN.15:= P3_Srobovanie.PAR.K40_AtlasCopcoInputs[4].23;
//    P3_Srobovanie.STAV.K40_Moment_ToleranciaMIN.16:= P3_Srobovanie.PAR.K40_AtlasCopcoInputs[4].8;
//    P3_Srobovanie.STAV.K40_Moment_ToleranciaMIN.17:= P3_Srobovanie.PAR.K40_AtlasCopcoInputs[4].9;
//    P3_Srobovanie.STAV.K40_Moment_ToleranciaMIN.18:= P3_Srobovanie.PAR.K40_AtlasCopcoInputs[4].10;
//    P3_Srobovanie.STAV.K40_Moment_ToleranciaMIN.19:= P3_Srobovanie.PAR.K40_AtlasCopcoInputs[4].11;
//    P3_Srobovanie.STAV.K40_Moment_ToleranciaMIN.20:= P3_Srobovanie.PAR.K40_AtlasCopcoInputs[4].12;
//    P3_Srobovanie.STAV.K40_Moment_ToleranciaMIN.21:= P3_Srobovanie.PAR.K40_AtlasCopcoInputs[4].13;
//    P3_Srobovanie.STAV.K40_Moment_ToleranciaMIN.22:= P3_Srobovanie.PAR.K40_AtlasCopcoInputs[4].14;
//    P3_Srobovanie.STAV.K40_Moment_ToleranciaMIN.23:= P3_Srobovanie.PAR.K40_AtlasCopcoInputs[4].15;
//    P3_Srobovanie.STAV.K40_Moment_ToleranciaMIN.24:= P3_Srobovanie.PAR.K40_AtlasCopcoInputs[4].0;
//    P3_Srobovanie.STAV.K40_Moment_ToleranciaMIN.25:= P3_Srobovanie.PAR.K40_AtlasCopcoInputs[4].1;
//    P3_Srobovanie.STAV.K40_Moment_ToleranciaMIN.26:= P3_Srobovanie.PAR.K40_AtlasCopcoInputs[4].2;
//    P3_Srobovanie.STAV.K40_Moment_ToleranciaMIN.27:= P3_Srobovanie.PAR.K40_AtlasCopcoInputs[4].3;
//    P3_Srobovanie.STAV.K40_Moment_ToleranciaMIN.28:= P3_Srobovanie.PAR.K40_AtlasCopcoInputs[4].4;
//    P3_Srobovanie.STAV.K40_Moment_ToleranciaMIN.29:= P3_Srobovanie.PAR.K40_AtlasCopcoInputs[4].5;
//    P3_Srobovanie.STAV.K40_Moment_ToleranciaMIN.30:= P3_Srobovanie.PAR.K40_AtlasCopcoInputs[4].6;
//    P3_Srobovanie.STAV.K40_Moment_ToleranciaMIN.31:= P3_Srobovanie.PAR.K40_AtlasCopcoInputs[4].7;
//    K40_Moment_ToleranciaMIN_REAL:= UDINT_TO_REAL(P3_Srobovanie.STAV.K40_Moment_ToleranciaMIN);
//    IF K40_Moment_ToleranciaMIN_REAL > 0 THEN
//      P3_Srobovanie.STAV.K40_Moment_ToleranciaMIN_REAL:= (K40_Moment_ToleranciaMIN_REAL*1.35)/65571;
//    ELSE
//        P3_Srobovanie.STAV.K40_Moment_ToleranciaMIN_REAL:=0.0;
//    END_IF

    K40_PrevodMomentu.AtlasMinimalnaTolerancia:=P3_Srobovanie.PAR.K40_AtlasCopcoInputs[4];
    P3_Srobovanie.STAV.K40_Moment_ToleranciaMIN_REAL:=K40_PrevodMomentu.ToleranciaMIN;

    (*P3_Srobovanie.STAV.K40_Moment_ToleranciaMIN_REAL:= K40_Moment_ToleranciaMIN_REAL /100;*)

    //Dosiahnutý úhol//
    P3_Srobovanie.STAV.K40_DosiahnutyUhol.0:= P3_Srobovanie.PAR.K40_AtlasCopcoInputs[0].24;
    P3_Srobovanie.STAV.K40_DosiahnutyUhol.1:= P3_Srobovanie.PAR.K40_AtlasCopcoInputs[0].25;
    P3_Srobovanie.STAV.K40_DosiahnutyUhol.2:= P3_Srobovanie.PAR.K40_AtlasCopcoInputs[0].26;
    P3_Srobovanie.STAV.K40_DosiahnutyUhol.3:= P3_Srobovanie.PAR.K40_AtlasCopcoInputs[0].27;
    P3_Srobovanie.STAV.K40_DosiahnutyUhol.4:= P3_Srobovanie.PAR.K40_AtlasCopcoInputs[0].28;
    P3_Srobovanie.STAV.K40_DosiahnutyUhol.5:= P3_Srobovanie.PAR.K40_AtlasCopcoInputs[0].29;
    P3_Srobovanie.STAV.K40_DosiahnutyUhol.6:= P3_Srobovanie.PAR.K40_AtlasCopcoInputs[0].30;
    P3_Srobovanie.STAV.K40_DosiahnutyUhol.7:= P3_Srobovanie.PAR.K40_AtlasCopcoInputs[0].31;
    P3_Srobovanie.STAV.K40_DosiahnutyUhol.8:= P3_Srobovanie.PAR.K40_AtlasCopcoInputs[0].16;
    P3_Srobovanie.STAV.K40_DosiahnutyUhol.9:= P3_Srobovanie.PAR.K40_AtlasCopcoInputs[0].17;
    P3_Srobovanie.STAV.K40_DosiahnutyUhol.10:= P3_Srobovanie.PAR.K40_AtlasCopcoInputs[0].18;
    P3_Srobovanie.STAV.K40_DosiahnutyUhol.11:= P3_Srobovanie.PAR.K40_AtlasCopcoInputs[0].19;
    P3_Srobovanie.STAV.K40_DosiahnutyUhol.12:= P3_Srobovanie.PAR.K40_AtlasCopcoInputs[0].20;
    P3_Srobovanie.STAV.K40_DosiahnutyUhol.13:= P3_Srobovanie.PAR.K40_AtlasCopcoInputs[0].21;
    P3_Srobovanie.STAV.K40_DosiahnutyUhol.14:= P3_Srobovanie.PAR.K40_AtlasCopcoInputs[0].22;
    P3_Srobovanie.STAV.K40_DosiahnutyUhol.15:= P3_Srobovanie.PAR.K40_AtlasCopcoInputs[0].23;

    //Uhol - Tolerancia MAX//
    P3_Srobovanie.STAV.K40_Uhol_ToleranciaMAX.0:= P3_Srobovanie.PAR.K40_AtlasCopcoInputs[2].8;
    P3_Srobovanie.STAV.K40_Uhol_ToleranciaMAX.1:= P3_Srobovanie.PAR.K40_AtlasCopcoInputs[2].9;
    P3_Srobovanie.STAV.K40_Uhol_ToleranciaMAX.2:= P3_Srobovanie.PAR.K40_AtlasCopcoInputs[2].10;
    P3_Srobovanie.STAV.K40_Uhol_ToleranciaMAX.3:= P3_Srobovanie.PAR.K40_AtlasCopcoInputs[2].11;
    P3_Srobovanie.STAV.K40_Uhol_ToleranciaMAX.4:= P3_Srobovanie.PAR.K40_AtlasCopcoInputs[2].12;
    P3_Srobovanie.STAV.K40_Uhol_ToleranciaMAX.5:= P3_Srobovanie.PAR.K40_AtlasCopcoInputs[2].13;
    P3_Srobovanie.STAV.K40_Uhol_ToleranciaMAX.6:= P3_Srobovanie.PAR.K40_AtlasCopcoInputs[2].14;
    P3_Srobovanie.STAV.K40_Uhol_ToleranciaMAX.7:= P3_Srobovanie.PAR.K40_AtlasCopcoInputs[2].15;
    P3_Srobovanie.STAV.K40_Uhol_ToleranciaMAX.8:= P3_Srobovanie.PAR.K40_AtlasCopcoInputs[2].0;
    P3_Srobovanie.STAV.K40_Uhol_ToleranciaMAX.9:= P3_Srobovanie.PAR.K40_AtlasCopcoInputs[2].1;
    P3_Srobovanie.STAV.K40_Uhol_ToleranciaMAX.10:= P3_Srobovanie.PAR.K40_AtlasCopcoInputs[2].2;
    P3_Srobovanie.STAV.K40_Uhol_ToleranciaMAX.11:= P3_Srobovanie.PAR.K40_AtlasCopcoInputs[2].3;
    P3_Srobovanie.STAV.K40_Uhol_ToleranciaMAX.12:= P3_Srobovanie.PAR.K40_AtlasCopcoInputs[2].4;
    P3_Srobovanie.STAV.K40_Uhol_ToleranciaMAX.13:= P3_Srobovanie.PAR.K40_AtlasCopcoInputs[2].5;
    P3_Srobovanie.STAV.K40_Uhol_ToleranciaMAX.14:= P3_Srobovanie.PAR.K40_AtlasCopcoInputs[2].6;
    P3_Srobovanie.STAV.K40_Uhol_ToleranciaMAX.15:= P3_Srobovanie.PAR.K40_AtlasCopcoInputs[2].7;

    //Uhol - Tolerancia MIN//
    P3_Srobovanie.STAV.K40_Uhol_ToleranciaMIN.0:= P3_Srobovanie.PAR.K40_AtlasCopcoInputs[2].24;
    P3_Srobovanie.STAV.K40_Uhol_ToleranciaMIN.1:= P3_Srobovanie.PAR.K40_AtlasCopcoInputs[2].25;
    P3_Srobovanie.STAV.K40_Uhol_ToleranciaMIN.2:= P3_Srobovanie.PAR.K40_AtlasCopcoInputs[2].26;
    P3_Srobovanie.STAV.K40_Uhol_ToleranciaMIN.3:= P3_Srobovanie.PAR.K40_AtlasCopcoInputs[2].27;
    P3_Srobovanie.STAV.K40_Uhol_ToleranciaMIN.4:= P3_Srobovanie.PAR.K40_AtlasCopcoInputs[2].28;
    P3_Srobovanie.STAV.K40_Uhol_ToleranciaMIN.5:= P3_Srobovanie.PAR.K40_AtlasCopcoInputs[2].29;
    P3_Srobovanie.STAV.K40_Uhol_ToleranciaMIN.6:= P3_Srobovanie.PAR.K40_AtlasCopcoInputs[2].30;
    P3_Srobovanie.STAV.K40_Uhol_ToleranciaMIN.7:= P3_Srobovanie.PAR.K40_AtlasCopcoInputs[2].31;
    P3_Srobovanie.STAV.K40_Uhol_ToleranciaMIN.8:= P3_Srobovanie.PAR.K40_AtlasCopcoInputs[2].16;
    P3_Srobovanie.STAV.K40_Uhol_ToleranciaMIN.9:= P3_Srobovanie.PAR.K40_AtlasCopcoInputs[2].17;
    P3_Srobovanie.STAV.K40_Uhol_ToleranciaMIN.10:= P3_Srobovanie.PAR.K40_AtlasCopcoInputs[2].18;
    P3_Srobovanie.STAV.K40_Uhol_ToleranciaMIN.11:= P3_Srobovanie.PAR.K40_AtlasCopcoInputs[2].19;
    P3_Srobovanie.STAV.K40_Uhol_ToleranciaMIN.12:= P3_Srobovanie.PAR.K40_AtlasCopcoInputs[2].20;
    P3_Srobovanie.STAV.K40_Uhol_ToleranciaMIN.13:= P3_Srobovanie.PAR.K40_AtlasCopcoInputs[2].21;
    P3_Srobovanie.STAV.K40_Uhol_ToleranciaMIN.14:= P3_Srobovanie.PAR.K40_AtlasCopcoInputs[2].22;
    P3_Srobovanie.STAV.K40_Uhol_ToleranciaMIN.15:= P3_Srobovanie.PAR.K40_AtlasCopcoInputs[2].23;

END_ACTION
```

#### OvlSkrutkovacichSetov.st
```iecst
ACTION OvlSkrutkovacichSetov:

		//***********************************Skrutkovací set K40************************************//
	//Volanie funkcie SequenceControl//
	SequenceControl(SC:= SC_SkrutkovaciSet_K40);

	CASE SC_SkrutkovaciSet_K40.Step OF

		0:
			SC_SkrutkovaciSet_K40.StepName:='0 - Nulovanie';
			P3_Srobovanie.SkrutSet_K40.Cmd.AutomatStart:= FALSE;
			P3_Srobovanie.SkrutSet_K40.Cmd.ManualStartHrniec:= FALSE;
			P3_Srobovanie.SkrutSet_K40.Cmd.PodajSkrutku:= FALSE;
			P3_Srobovanie.CMD.RR_SkrutSetK40_PodajSkrutku:= FALSE;
			P3_Srobovanie.CMD.RR_SkrutSetK40_Zasobnik_RUN:= FALSE;
			P3_Srobovanie.CMD.RR_SkrutSetK40_VysunBrzdu:= FALSE;
			P3_Srobovanie.SkrutSet_K40.Cmd.ManualPresunBrzdu:= FALSE;
			P3_Srobovanie.STAV.SkrutkaK40_READY:= FALSE;

			IF SC_P3_Srobovanie.Step <> 0 THEN
				SC_SkrutkovaciSet_K40.ResetStep:= TRUE;
				SC_SkrutkovaciSet_K40.Step:= 1;
			END_IF

		1:
			SC_SkrutkovaciSet_K40.StepName:='1 - Rozhodnutie o cinnosti';

			IF P3_Srobovanie.Automat THEN
				SC_SkrutkovaciSet_K40.ResetStep:= TRUE;
				SC_SkrutkovaciSet_K40.Step:= 10;
			ELSIF P3_Srobovanie.Manual THEN
				SC_SkrutkovaciSet_K40.ResetStep:= TRUE;
				SC_SkrutkovaciSet_K40.Step:= 20;
			END_IF

		10:
			SC_SkrutkovaciSet_K40.StepName:='10 - Automaticky rezim - cakam na signal podaj skrutku';
			SC_SkrutkovaciSet_K40.IdleTime.PT:= T#2s;
			SC_SkrutkovaciSet_K40.AlarmTime.PT:= T#5s;

			P3_Srobovanie.SkrutSet_K40.Cmd.AutomatStart:= TRUE;

			IF P3_Srobovanie.CMD.PodajSkrutku_K40 THEN
				P3_Srobovanie.CMD.PodajSkrutku_K40:= FALSE;
				SC_SkrutkovaciSet_K40.ResetStep:= TRUE;
				SC_SkrutkovaciSet_K40.Step:= 13;
			END_IF

		13:
			SC_SkrutkovaciSet_K40.StepName:='13 - Automaticky rezim - podanie skrutky do skrutkovacky';
			SC_SkrutkovaciSet_K40.IdleTime.PT:= T#2s;
			SC_SkrutkovaciSet_K40.AlarmTime.PT:= T#5s;

			IF NOT SC_SkrutkovaciSet_K40.Switch1 THEN
				P3_Srobovanie.SkrutSet_K40.Cmd.PodajSkrutku:= TRUE;
				SC_SkrutkovaciSet_K40.Switch1:= TRUE;
			END_IF

			IF P3_Srobovanie.SkrutSet_K40.Status.SkrutkaPripravena THEN
				P3_Srobovanie.STAV.SkrutkaK40_READY:= TRUE;
				P3_Srobovanie.SkrutSet_K40.Cmd.PodajSkrutku:= FALSE;
				SC_SkrutkovaciSet_K40.ResetStep:= TRUE;
				SC_SkrutkovaciSet_K40.Step:= 15;
			ELSIF P3_Srobovanie.SkrutSet_K40.Error.ErrorBit THEN
				P3_Srobovanie.SkrutSet_K40.Cmd.PodajSkrutku:= FALSE;
				P34_Alarmy[328]:= TRUE;
				P3_Pracovisko.STAV.Porucha_ST1:= TRUE;
			END_IF

		15:
			SC_SkrutkovaciSet_K40.StepName:='15 - Automaticky rezim - cakam na zrusenie stavu skrutka K40 READY';
			SC_SkrutkovaciSet_K40.IdleTime.PT:= T#2s;
			SC_SkrutkovaciSet_K40.AlarmTime.PT:= T#5s;

			IF NOT P3_Srobovanie.STAV.SkrutkaK40_READY THEN
				SC_SkrutkovaciSet_K40.ResetStep:= TRUE;
				SC_SkrutkovaciSet_K40.Step:= 10;
			ELSIF P3_Srobovanie.Manual THEN
				P3_Srobovanie.SkrutSet_K40.Cmd.AutomatStart:= FALSE;
				SC_SkrutkovaciSet_K40.ResetStep:= TRUE;
				SC_SkrutkovaciSet_K40.Step:= 20;
			END_IF

		20:
			SC_SkrutkovaciSet_K40.StepName:='20 - Manualny rezim';
			SC_SkrutkovaciSet_K40.IdleTime.PT:= T#2s;
			SC_SkrutkovaciSet_K40.AlarmTime.PT:= T#5s;

			//Ovládanie zásobníka//
			IF P3_Srobovanie.CMD.RR_SkrutSetK40_Zasobnik_RUN THEN
				P3_Srobovanie.SkrutSet_K40.Cmd.AutomatStart:= FALSE;
				P3_Srobovanie.SkrutSet_K40.Cmd.ManualStartHrniec:= TRUE;
			ELSE
				P3_Srobovanie.SkrutSet_K40.Cmd.ManualStartHrniec:= FALSE;
			END_IF

			//Ovládanie brzdy//
			IF P3_Srobovanie.CMD.RR_SkrutSetK40_VysunBrzdu THEN
				P3_Srobovanie.SkrutSet_K40.Cmd.AutomatStart:= FALSE;
				P3_Srobovanie.SkrutSet_K40.Cmd.ManualPresunBrzdu:= TRUE;
			ELSE
				P3_Srobovanie.SkrutSet_K40.Cmd.ManualPresunBrzdu:= FALSE;
			END_IF

			//Podanie skrutky//
			IF P3_Srobovanie.CMD.RR_SkrutSetK40_PodajSkrutku THEN
				P3_Srobovanie.CMD.RR_SkrutSetK40_PodajSkrutku:= FALSE;
				P3_Srobovanie.CMD.RR_SkrutSetK40_Zasobnik_RUN:= FALSE;
				P3_Srobovanie.SkrutSet_K40.Cmd.ManualStartHrniec:= FALSE;
				P3_Srobovanie.SkrutSet_K40.Cmd.ManualPresunBrzdu:= FALSE;
				P3_Srobovanie.CMD.PodajSkrutku_K40:= TRUE;
				SC_SkrutkovaciSet_K40.ResetStep:= TRUE;
				SC_SkrutkovaciSet_K40.Step:= 10;
			END_IF

	END_CASE

	//***********************************Skrutkovací set M5***************************************//
	//Volanie funkcie SequenceControl//
	SequenceControl(SC:= SC_SkrutkovaciSet_M5);

	CASE SC_SkrutkovaciSet_M5.Step OF

		0:
			SC_SkrutkovaciSet_M5.StepName:='0 - Nulovanie';
			P3_Srobovanie.SkrutSet_M5.CMD.ENABLE:= FALSE;
			P3_Srobovanie.SkrutSet_M5.CMD.RucnyRezim:= FALSE;
			P3_Srobovanie.SkrutSet_M5.CMD.PodajSkrutku:= FALSE;
			P3_Srobovanie.SkrutSet_M5.CMD.RR_OtocPodavac_Vstup:= FALSE;
			P3_Srobovanie.SkrutSet_M5.CMD.RR_OtocPodavac_Vystup:= FALSE;
			P3_Srobovanie.SkrutSet_M5.CMD.RR_ZapniVibrolistu:= FALSE;
			P3_Srobovanie.SkrutSet_M5.CMD.RR_ZapniZasobnik:= FALSE;

			IF SC_P3_Srobovanie.Step <> 0 THEN
				SC_SkrutkovaciSet_M5.ResetStep:= TRUE;
				SC_SkrutkovaciSet_M5.Step:= 1;
			END_IF

		1:
			SC_SkrutkovaciSet_M5.StepName:='1 - Rozhodnutie o cinnosti';

			IF P3_Srobovanie.Automat THEN
				SC_SkrutkovaciSet_M5.ResetStep:= TRUE;
				SC_SkrutkovaciSet_M5.Step:= 10;
			ELSIF P3_Srobovanie.Manual THEN
				SC_SkrutkovaciSet_M5.ResetStep:= TRUE;
				SC_SkrutkovaciSet_M5.Step:= 20;
			END_IF

		10:
			SC_SkrutkovaciSet_M5.StepName:='10 - Automaticky rezim - cakam na signal podaj skrutku';
			SC_SkrutkovaciSet_M5.IdleTime.PT:= T#2s;
			SC_SkrutkovaciSet_M5.AlarmTime.PT:= T#5s;

			P3_Srobovanie.SkrutSet_M5.CMD.ENABLE:= TRUE;

			IF P3_Srobovanie.CMD.PodajSkrutku_M5 THEN
				P3_Srobovanie.CMD.PodajSkrutku_M5:= FALSE;
				SC_SkrutkovaciSet_M5.ResetStep:= TRUE;
				SC_SkrutkovaciSet_M5.Step:= 13;
			END_IF

		13:
			SC_SkrutkovaciSet_M5.StepName:='13 - Automaticky rezim - podanie skrutky';
			SC_SkrutkovaciSet_M5.IdleTime.PT:= T#2s;
			SC_SkrutkovaciSet_M5.AlarmTime.PT:= T#5s;

			IF NOT SC_SkrutkovaciSet_M5.Switch1 THEN
				P3_Srobovanie.SkrutSet_M5.CMD.PodajSkrutku:= TRUE;
				SC_SkrutkovaciSet_M5.Switch1:= TRUE;
			END_IF

			IF P3_Srobovanie.SkrutSet_M5.STAV.SkrutkaPripravena THEN
				P3_Srobovanie.SkrutSet_M5.CMD.PodajSkrutku:= FALSE;
				SC_SkrutkovaciSet_M5.ResetStep:= TRUE;
				SC_SkrutkovaciSet_M5.Step:= 15;
			ELSIF P3_Srobovanie.SkrutSet_M5.STAV.ERROR THEN
				P3_Srobovanie.SkrutSet_M5.CMD.PodajSkrutku:= FALSE;
				P34_Alarmy[327]:= TRUE;
				P3_Pracovisko.STAV.Porucha_ST1:= TRUE;
			END_IF

		15:
			SC_SkrutkovaciSet_M5.StepName:='15 - Automaticky rezim - ukoncenie podania skrutky M5';
			SC_SkrutkovaciSet_M5.IdleTime.PT:= T#2s;
			SC_SkrutkovaciSet_M5.AlarmTime.PT:= T#5s;

			IF P3_Srobovanie.Manual THEN
				SC_SkrutkovaciSet_M5.ResetStep:= TRUE;
				SC_SkrutkovaciSet_M5.Step:= 20;
			ELSE
				SC_SkrutkovaciSet_M5.ResetStep:= TRUE;
				SC_SkrutkovaciSet_M5.Step:= 10;
			END_IF

		20:
			SC_SkrutkovaciSet_M5.StepName:='20 - Manualny rezim';
			SC_SkrutkovaciSet_M5.IdleTime.PT:= T#2s;
			SC_SkrutkovaciSet_M5.AlarmTime.PT:= T#5s;

			P3_Srobovanie.SkrutSet_M5.CMD.ENABLE:= TRUE;
			P3_Srobovanie.SkrutSet_M5.CMD.RucnyRezim:= TRUE;

			//Ovládanie zásobníka//
			IF P3_Srobovanie.CMD.RR_SkrutSetM5_Zasobnik_RUN THEN
				P3_Srobovanie.SkrutSet_M5.CMD.RR_ZapniZasobnik:= TRUE;
			ELSE
				P3_Srobovanie.SkrutSet_M5.CMD.RR_ZapniZasobnik:= FALSE;
			END_IF

			//Ovládanie vibrolišty//
			IF P3_Srobovanie.CMD.RR_SkrutSetM5_Vibrolista_RUN THEN
				P3_Srobovanie.SkrutSet_M5.CMD.RR_ZapniVibrolistu:= TRUE;
			ELSE
				P3_Srobovanie.SkrutSet_M5.CMD.RR_ZapniVibrolistu:= FALSE;
			END_IF

			//Otáčanie podavača skrutiek//
			IF P3_Srobovanie.CMD.RR_SkrutSetM5_OtocPodavac_Vstup THEN
				P3_Srobovanie.SkrutSet_M5.CMD.RR_OtocPodavac_Vstup:= TRUE;
				P3_Srobovanie.CMD.RR_SkrutSetM5_OtocPodavac_Vstup:= FALSE;
			ELSIF P3_Srobovanie.CMD.RR_SkrutSetM5_OtocPodavac_Vystup THEN
				P3_Srobovanie.SkrutSet_M5.CMD.RR_OtocPodavac_Vystup:= TRUE;
				P3_Srobovanie.CMD.RR_SkrutSetM5_OtocPodavac_Vystup:= FALSE;
			END_IF

			//Podanie skrutky//
			IF P3_Srobovanie.CMD.RR_SkrutSetM5_PodajSkrutku THEN
				P3_Srobovanie.CMD.RR_SkrutSetM5_PodajSkrutku:= FALSE;
				P3_Srobovanie.CMD.RR_SkrutSetM5_Zasobnik_RUN:= FALSE;
				P3_Srobovanie.CMD.RR_SkrutSetM5_Vibrolista_RUN:= FALSE;
				P3_Srobovanie.SkrutSet_M5.CMD.RucnyRezim:= TRUE;
				P3_Srobovanie.CMD.PodajSkrutku_M5:= TRUE;
				SC_SkrutkovaciSet_M5.ResetStep:= TRUE;
				SC_SkrutkovaciSet_M5.Step:= 10;
			END_IF

	END_CASE

END_ACTION
```

### Program Logical/Program/Pracovisko_3/P3_HV_Test (IEC)

#### Main.st - Init, cyclic, exit code
```iecst
PROGRAM _INIT

	 P3_HV_Test.PAR.CisloPortuKlienta:= 1031;

END_PROGRAM

PROGRAM _CYCLIC

	//Volanie funkcie SequenceControl//
	SequenceControl(SC:= SC_P3_HV_Test);

	//Volanie podprogramov//
	OvlCentrovacky;
	OvlHornychKontaktov;
	OvlSpodnychKontaktov;
	IOLinkKomunikacia;
	COM_Tester;

	//Reset sekcie //
	IF P3_HV_Test.Reset THEN
		SC_P3_HV_Test.Step:= 0;
		P3_HV_Test.Reset:= FALSE;
	ELSIF NOT Safety.STAV.Linka_ZonaCS_AKTIVNA THEN
		SC_P3_HV_Test.Step:= 0;
	END_IF

	CASE SC_P3_HV_Test.Step OF

		0:
			SC_P3_HV_Test.StepName:='0 - Nulovanie';
			SC_OvlCentrovacky.Step:= 0;
			SC_OvlHornychKontaktov.Step:= 0;
			SC_OvlSpodnychKontaktov.Step:= 0;
			SC_OvlTesteraHV.Step:= 0;
			P3_HV_Test.Automat:= FALSE;
			P3_HV_Test.KoniecCyklu:= FALSE;
			P3_HV_Test.Manual:= FALSE;
			P3_HV_Test.STAV.PoINIT:= FALSE;
			P3_HV_Test.OUT.ZasunStoper:= FALSE;
			P3_HV_Test.OUT.PritlacenieKontaktovTestera_ON:= FALSE;
			P3_HV_Test.OUT.PruzenieHornychKontaktov_VYSUN:= FALSE;
			P3_HV_Test.OUT.PruzenieHornychKontaktov_ZASUN:= TRUE;
			P3_HV_Test.OUT.HorneKontakty_VYSUN:= FALSE;
			P3_HV_Test.OUT.HorneKontakty_ZASUN:= TRUE;
			P3_HV_Test.OUT.SpodneKontakty_VYSUN:= FALSE;
			P3_HV_Test.OUT.SpodneKontakty_ZASUN:= TRUE;
			P3_HV_Test.RFID_hlava.PrecitajChipRFID:= FALSE;
			P3_HV_Test.CMD.RR_ZatvorTester:= FALSE;
			P3_HV_Test.CMD.StartTestovania:= FALSE;
			P3_HV_Test.CMD.RR_VysunPruzenieKontaktov:= FALSE;
			P3_HV_Test.STAV.RR_SekvenciaTestera_BUSY:= FALSE;
			P3_HV_Test.CMD.OpatovnyTest:= FALSE;
			P34_Vizu.ZobrazHL1_HVtest:= FALSE;
			P3_StoperSrobovania.STAV.PrebiehaVyvezeniePaletky:= FALSE;
			P3_HV_Test.STAV.PrebiehaVyvezeniePaletky:= FALSE;
			P3_HV_Test.STAV.PaletkaOznacena_NG:= FALSE;
			TestovaciKus:= FALSE;
			P3_HVtest_Taktime.IN.START_MeraniaCasu:= FALSE;
			P3_HVtest_Taktime.IN.START_MeraniaStratovehoCasu:= FALSE;

			PocetDopytovNaTester:= 0;

			IF Safety.STAV.Linka_ZonaCS_AKTIVNA AND
				Safety.STAV.P3_ZonaBunky_AKTIVNA AND
				P3_Pracovisko.STAV.HardwareBunky_OK AND
				NOT P3_Pracovisko.STAV.Porucha_ST1 AND
				NOT P3_Pracovisko.STAV.Porucha_ST2 AND
				NOT P3_Pracovisko.STAV.Porucha_ST3 AND
				NOT P3_Pracovisko.STAV.Porucha_ST4 AND
				NOT P3_Pracovisko.STAV.Porucha_ST5 AND
				NOT P3_Pracovisko.STAV.Porucha_ST6 AND
				NOT P3_Pracovisko.STAV.Porucha_ST7 AND
				NOT P3_Pracovisko.STAV.Porucha_ST8 THEN
				SC_P3_HV_Test.ResetStep:= TRUE;
				SC_P3_HV_Test.Step:= 1;
			END_IF

		1:
			SC_P3_HV_Test.StepName:='1 - Cakam na spustenie vyroby';
			P3_HV_Test.KoniecCyklu:= FALSE;
			IF P3_HV_Test.Automat THEN
				SC_P3_HV_Test.Step:= 2;
			ELSIF P3_HV_Test.Manual THEN
				SC_P3_HV_Test.Step:= 700;
			END_IF

			//********************************************************Inicializácia****************************************************************************//

		2:
			SC_P3_HV_Test.StepName:='2 - Inicializacia - cakam na spustenie inicializacie';
			SC_P3_HV_Test.IdleTime.PT:= T#500ms;
			SC_P3_HV_Test.AlarmTime.PT:= T#5s;

			SC_P3_HV_Test.IdleTime.IN:= TRUE;

			IF SC_P3_HV_Test.IdleTime.Q THEN
				SC_P3_HV_Test.ResetStep:= TRUE;
				SC_P3_HV_Test.Step:= 5;
			END_IF

		5:
			SC_P3_HV_Test.StepName:='5 - Inicializacia - zasunutie spodnych kontaktov';
			SC_P3_HV_Test.IdleTime.PT:= T#4s;
			SC_P3_HV_Test.AlarmTime.PT:= T#5s;

			IF NOT SC_P3_HV_Test.Switch1 THEN
				SpodneKontakty_ZASUN:= TRUE;
				SC_P3_HV_Test.Switch1:= TRUE;
			END_IF

			IF P3_HV_Test.IN.SpodneKontakty_ZASUNUTE THEN
				SC_P3_HV_Test.ResetStep:= TRUE;
				SC_P3_HV_Test.Step:= 8;
			END_IF

		8:
			SC_P3_HV_Test.StepName:='8 - Inicializacia - zasunutie hornych kontaktov';
			SC_P3_HV_Test.IdleTime.PT:= T#4s;
			SC_P3_HV_Test.AlarmTime.PT:= T#5s;

			IF NOT SC_P3_HV_Test.Switch1 THEN
				HorneKontakty_ZASUN:= TRUE;
				SC_P3_HV_Test.Switch1:= TRUE;
			END_IF

			IF P3_HV_Test.IN.HorneKontakty_ZASUNUTE THEN
				SC_P3_HV_Test.ResetStep:= TRUE;
				SC_P3_HV_Test.Step:= 10;
			END_IF

		10:
			SC_P3_HV_Test.StepName:='10 - Inicializacia - zasunutie cenrovacky';
			SC_P3_HV_Test.IdleTime.PT:= T#4s;
			SC_P3_HV_Test.AlarmTime.PT:= T#5s;

			IF NOT SC_P3_HV_Test.Switch1 THEN
				Centrovacku_ZASUN:= TRUE;
				SC_P3_HV_Test.Switch1:= TRUE;
			END_IF

			IF P3_HV_Test.IN.Centrovanie_ZASUNUTE THEN
				SC_P3_HV_Test.ResetStep:= TRUE;
				SC_P3_HV_Test.Step:= 13;
			END_IF

		13:
			SC_P3_HV_Test.StepName:='13 - Inicializacia - kontrola kontaktov HV testu';
			SC_P3_HV_Test.IdleTime.PT:= T#4s;
			SC_P3_HV_Test.AlarmTime.PT:= T#5s;

			IF Linka.PAR.ZvolenyModel = '4F' AND P3_HV_Test.IN.TypKonektoru_4F THEN
				SC_P3_HV_Test.ResetStep:= TRUE;
				SC_P3_HV_Test.Step:= 15;
			ELSIF Linka.PAR.ZvolenyModel = '5F' AND P3_HV_Test.IN.TypKonektoru_5F_5H THEN
				SC_P3_HV_Test.ResetStep:= TRUE;
				SC_P3_HV_Test.Step:= 15;
			ELSIF Linka.PAR.ZvolenyModel = '5H' AND P3_HV_Test.IN.TypKonektoru_5F_5H THEN
				SC_P3_HV_Test.ResetStep:= TRUE;
				SC_P3_HV_Test.Step:= 15;
			ELSE
				P34_Alarmy[326]:= TRUE;
				P3_Pracovisko.STAV.Porucha_ST2:= TRUE;
			END_IF

		15:
			SC_P3_HV_Test.StepName:='15 - Inicializacia - hladanie paletky';
			SC_P3_HV_Test.IdleTime.PT:= T#5s;
			SC_P3_HV_Test.AlarmTime.PT:= T#5s;

			SC_P3_HV_Test.IdleTime.IN:= P3_Dopravniky.STAV.PoINIT;

			IF P3_HV_Test.RFID_hlava.PritomnostPaletky THEN
				SC_P3_HV_Test.ResetStep:= TRUE;
				SC_P3_HV_Test.Step:= 20;
			ELSIF SC_P3_HV_Test.IdleTime.Q THEN
				P3_HV_Test.STAV.PoINIT:= TRUE;
				SC_P3_HV_Test.ResetStep:= TRUE;
				SC_P3_HV_Test.Step:= 100;
			END_IF

		20:
			SC_P3_HV_Test.StepName:='20 - Inicializacia - precitanie cisla paletky';
			SC_P3_HV_Test.IdleTime.PT:= T#200ms;
			SC_P3_HV_Test.AlarmTime.PT:= T#5s;

			SC_P3_HV_Test.IdleTime.IN:= P3_HV_Test.RFID_hlava.PritomnostPaletky;

			IF SC_P3_HV_Test.IdleTime.Q AND NOT SC_P3_HV_Test.Switch1 THEN
				P3_HV_Test.RFID_hlava.PrecitajChipRFID:= TRUE;
				i:= 0;
				SC_P3_HV_Test.Switch1:= TRUE;
			END_IF

			IF P3_HV_Test.RFID_hlava.Stav_CitanieZapis_OK AND P3_HV_Test.RFID_hlava.PrecitaneCisloPaletky <> 0 THEN
				i:= P3_HV_Test.RFID_hlava.PrecitaneCisloPaletky;
				P3_HV_Test.RFID_hlava.PrecitajChipRFID:= FALSE;
				SC_P3_HV_Test.ResetStep:= TRUE;
				SC_P3_HV_Test.Step:= 23;
			END_IF

		23:
			SC_P3_HV_Test.StepName:='23 - Inicializacia - priradenie indexu paletky na zaklade precitanej hodnoty';
			SC_P3_HV_Test.IdleTime.PT:= T#200ms;
			SC_P3_HV_Test.AlarmTime.PT:= T#5s;

			IF i<> 0 THEN
				P3_HV_Test.PAR.CisloPaletky_STRING:= USINT_TO_STRING(i);
				Paletka[i].PAR.CisloPaletky:= USINT_TO_STRING(i);
				SC_P3_HV_Test.ResetStep:= TRUE;
				SC_P3_HV_Test.Step:= 30;
			ELSE
				P34_Alarmy[366]:= TRUE;
				P3_Pracovisko.STAV.Porucha_ST2:= TRUE;
			END_IF

		30:
			SC_P3_HV_Test.StepName:='30 - Inicializacia - kontrola stavu paletky';
			SC_P3_HV_Test.IdleTime.PT:= T#200ms;
			SC_P3_HV_Test.AlarmTime.PT:= T#5s;

			IF Paletka[i].STAV.StavPaletky = '' THEN
				Paletka[i].STAV.StavPaletky:= 'NG';
				SC_P3_HV_Test.ResetStep:= TRUE;
				SC_P3_HV_Test.Step:= 560;
			ELSIF Paletka[i].STAV.StavPaletky = 'PRECH' THEN
				P3_HV_Test.STAV.PoINIT:= TRUE;
				SC_P3_HV_Test.ResetStep:= TRUE;
				SC_P3_HV_Test.Step:= 560;
			ELSIF Paletka[i].STAV.StavPaletky = 'TEST' AND Paletka[i].STAV.CisloTestovacejStanice = 'ST_7' THEN
				TestovaciKus:= TRUE;
				P3_HV_Test.STAV.PoINIT:= TRUE;
				SC_P3_HV_Test.ResetStep:= TRUE;
				SC_P3_HV_Test.Step:= 110;
			ELSIF Paletka[i].STAV.StavPaletky = 'TEST' AND Paletka[i].STAV.CisloTestovacejStanice <> 'ST_7' THEN
				P3_HV_Test.STAV.PoINIT:= TRUE;
				SC_P3_HV_Test.ResetStep:= TRUE;
				SC_P3_HV_Test.Step:= 560;
			ELSIF Paletka[i].STAV.StavPaletky = 'REV' AND Paletka[i].STAV.CisloRevorkovejStanice = 'ST_7_HV' THEN
				P3_HV_Test.STAV.PoINIT:= TRUE;
				SC_P3_HV_Test.ResetStep:= TRUE;
				SC_P3_HV_Test.Step:= 110;
			ELSIF Paletka[i].STAV.StavPaletky = 'REV' AND Paletka[i].STAV.CisloRevorkovejStanice <> 'ST_7_HV' THEN
				P3_HV_Test.STAV.PoINIT:= TRUE;
				SC_P3_HV_Test.ResetStep:= TRUE;
				SC_P3_HV_Test.Step:= 560;
			ELSIF Paletka[i].STAV.StavPaletky = 'OK' THEN
				SC_P3_HV_Test.ResetStep:= TRUE;
				SC_P3_HV_Test.Step:= 33;
			ELSIF Paletka[i].STAV.StavPaletky = 'NG' THEN
				P3_HV_Test.STAV.PoINIT:= TRUE;
				SC_P3_HV_Test.ResetStep:= TRUE;
				SC_P3_HV_Test.Step:= 560;
			END_IF

		33:
			SC_P3_HV_Test.StepName:='33 - Inicializacia - kontrola ukonceneho HV testu';
			SC_P3_HV_Test.IdleTime.PT:= T#200ms;
			SC_P3_HV_Test.AlarmTime.PT:= T#5s;

			IF Paletka[i].STAV.HV_Test_Ukonceny THEN
				P3_HV_Test.STAV.PoINIT:= TRUE;
				SC_P3_HV_Test.ResetStep:= TRUE;
				SC_P3_HV_Test.Step:= 560;
			ELSE
				P3_HV_Test.STAV.PoINIT:= TRUE;
				SC_P3_HV_Test.ResetStep:= TRUE;
				SC_P3_HV_Test.Step:= 110;
			END_IF

			//********************************************************Automatický režim****************************************************************************//

		100:
			SC_P3_HV_Test.StepName:='100 - Automaticky Rezim - cakam na príchod paletky na stoper';
			SC_P3_HV_Test.IdleTime.PT:= T#200ms;
			SC_P3_HV_Test.AlarmTime.PT:= T#5s;

			SC_P3_HV_Test.IdleTime.IN:= P3_HV_Test.RFID_hlava.PritomnostPaletky;

			IF P3_HV_Test.RFID_hlava.PritomnostPaletky THEN
				P3_StoperSrobovania.STAV.PrebiehaVyvezeniePaletky:= FALSE;
			END_IF

			IF NOT SC_P3_HV_Test.Switch1 AND P3_HV_Test.RFID_hlava.PritomnostPaletky THEN
				P3_HVtest_Taktime.IN.START_MeraniaCasu:= TRUE;
				P3_HVtest_Taktime.IN.ZAPIS_MeraniaCasu:= TRUE;
				P3_HVtest_Taktime.IN.ZAPIS_StratovyCas:= TRUE;
				Buffer_8.Hodnota:= P3_HVtest_Taktime.OUT.StratoveSekundy;
				Buffer_8.ZapisHodnotu:= TRUE;
				SC_P3_HV_Test.Switch1:= TRUE;
			END_IF

			IF P3_HV_Test.KoniecCyklu THEN
				SC_P3_HV_Test.ResetStep:= TRUE;
				SC_P3_HV_Test.Step:= 0;
			ELSIF SC_P3_HV_Test.IdleTime.Q THEN
				SC_P3_HV_Test.ResetStep:= TRUE;
				SC_P3_HV_Test.Step:= 101;
			END_IF

		101:
			SC_P3_HV_Test.StepName:='101 - Automaticky Rezim - precitanie cisla paletky';
			SC_P3_HV_Test.IdleTime.PT:= T#200ms;
			SC_P3_HV_Test.AlarmTime.PT:= T#5s;
			SC_P3_HV_Test.IdleTime.IN:= TRUE;

			IF NOT SC_P3_HV_Test.Switch1 THEN
				P3_HV_Test.RFID_hlava.PrecitajChipRFID:= TRUE;
				i:= 0;
				SC_P3_HV_Test.Switch1:= TRUE;
			END_IF

			IF P3_HV_Test.RFID_hlava.Stav_CitanieZapis_OK AND P3_HV_Test.RFID_hlava.PrecitaneCisloPaletky <> 0 THEN
				i:= P3_HV_Test.RFID_hlava.PrecitaneCisloPaletky;
				P3_HV_Test.RFID_hlava.PrecitajChipRFID:= FALSE;
				SC_P3_HV_Test.ResetStep:= TRUE;
				SC_P3_HV_Test.Step:= 102;
			END_IF

		102:
			SC_P3_HV_Test.StepName:='102 - Automaticky Rezim - priradenie indexu paletky na zaklade precitanej hodnoty';
			SC_P3_HV_Test.IdleTime.PT:= T#200ms;
			SC_P3_HV_Test.AlarmTime.PT:= T#5s;

			IF i<> 0 THEN
				P3_HV_Test.PAR.CisloPaletky_STRING:= USINT_TO_STRING(i);
				Paletka[i].PAR.CisloPaletky:= USINT_TO_STRING(i);
				SC_P3_HV_Test.ResetStep:= TRUE;
				SC_P3_HV_Test.Step:= 103;
			ELSE
				P34_Alarmy[366]:= TRUE;
				P3_Pracovisko.STAV.Porucha_ST2:= TRUE;
			END_IF

		103:
			SC_P3_HV_Test.StepName:='103 - Automaticky Rezim - kontrola stavu paletky';
			SC_P3_HV_Test.IdleTime.PT:= T#200ms;
			SC_P3_HV_Test.AlarmTime.PT:= T#5s;

			IF Paletka[i].STAV.StavPaletky = '' THEN
				Paletka[i].STAV.StavPaletky:= 'NG';
				SC_P3_HV_Test.ResetStep:= TRUE;
				SC_P3_HV_Test.Step:= 560;
			ELSIF Paletka[i].STAV.StavPaletky = 'PRECH' THEN
				SC_P3_HV_Test.ResetStep:= TRUE;
				SC_P3_HV_Test.Step:= 560;
			ELSIF Paletka[i].STAV.StavPaletky = 'TEST' AND Paletka[i].STAV.CisloTestovacejStanice = 'ST_7' THEN
				TestovaciKus:= TRUE;
				SC_P3_HV_Test.ResetStep:= TRUE;
				SC_P3_HV_Test.Step:= 110;
			ELSIF Paletka[i].STAV.StavPaletky = 'TEST' AND Paletka[i].STAV.CisloTestovacejStanice <> 'ST_7' THEN
				SC_P3_HV_Test.ResetStep:= TRUE;
				SC_P3_HV_Test.Step:= 560;
			ELSIF Paletka[i].STAV.StavPaletky = 'REV' AND Paletka[i].STAV.CisloRevorkovejStanice = 'ST_7_HV' THEN
				SC_P3_HV_Test.ResetStep:= TRUE;
				SC_P3_HV_Test.Step:= 110;
			ELSIF Paletka[i].STAV.StavPaletky = 'REV' AND Paletka[i].STAV.CisloRevorkovejStanice <> 'ST_7_HV' THEN
				SC_P3_HV_Test.ResetStep:= TRUE;
				SC_P3_HV_Test.Step:= 560;
			ELSIF Paletka[i].STAV.StavPaletky = 'OK' THEN
				SC_P3_HV_Test.ResetStep:= TRUE;
				SC_P3_HV_Test.Step:= 110;
			ELSIF Paletka[i].STAV.StavPaletky = 'NG' THEN
				SC_P3_HV_Test.ResetStep:= TRUE;
				SC_P3_HV_Test.Step:= 560;
			END_IF

			//Zatvorenie HV testera//

		110:
			SC_P3_HV_Test.StepName:='110 - Automaticky Rezim - zacentrovanie paletky';
			SC_P3_HV_Test.IdleTime.PT:= T#200ms;
			SC_P3_HV_Test.AlarmTime.PT:= T#5s;

			IF NOT SC_P3_HV_Test.Switch1 THEN
				Centrovacku_VYSUN:= TRUE;
				SC_P3_HV_Test.Switch1:= TRUE;
			END_IF

			IF P3_HV_Test.IN.Centrovanie_VYSUNUTE THEN
				SC_P3_HV_Test.ResetStep:= TRUE;
				SC_P3_HV_Test.Step:= 113;
			END_IF

		113:
			SC_P3_HV_Test.StepName:='113 - Automaticky Rezim - vysunutie pruzenia hornych kontaktov';
			SC_P3_HV_Test.IdleTime.PT:= T#300ms;
			SC_P3_HV_Test.AlarmTime.PT:= T#5s;

			IF NOT SC_P3_HV_Test.Switch1 THEN
				P3_HV_Test.OUT.PruzenieHornychKontaktov_ZASUN:= FALSE;
				P3_HV_Test.OUT.PruzenieHornychKontaktov_VYSUN:= TRUE;
				SC_P3_HV_Test.IdleTime.IN:= TRUE;
				SC_P3_HV_Test.Switch1:= TRUE;
			END_IF

			IF SC_P3_HV_Test.IdleTime.Q THEN
				SC_P3_HV_Test.ResetStep:= TRUE;
				SC_P3_HV_Test.Step:= 115;
			END_IF

		115:
			SC_P3_HV_Test.StepName:='115 - Automaticky Rezim - vysunutie hornych kontaktov';
			SC_P3_HV_Test.IdleTime.PT:= T#200ms;
			SC_P3_HV_Test.AlarmTime.PT:= T#5s;

			IF NOT SC_P3_HV_Test.Switch1 THEN
				HorneKontakty_VYSUN:= TRUE;
				SC_P3_HV_Test.Switch1:= TRUE;
			END_IF

			IF P3_HV_Test.IN.HorneKontakty_VYSUNUTE THEN
				SC_P3_HV_Test.ResetStep:= TRUE;
				SC_P3_HV_Test.Step:= 118;
			END_IF

		118:
			SC_P3_HV_Test.StepName:='118 - Automaticky Rezim - vysunutie spodnych kontaktov';
			SC_P3_HV_Test.IdleTime.PT:= T#200ms;
			SC_P3_HV_Test.AlarmTime.PT:= T#5s;

			IF NOT SC_P3_HV_Test.Switch1 THEN
				SpodneKontakty_VYSUN:= TRUE;
				SC_P3_HV_Test.Switch1:= TRUE;
			END_IF

			IF P3_HV_Test.IN.SpodneKontakty_VYSUNUTE THEN
				SC_P3_HV_Test.ResetStep:= TRUE;
				SC_P3_HV_Test.Step:= 120;
			END_IF

		120:
			SC_P3_HV_Test.StepName:='120 - Automaticky Rezim - pritlacenie kontaktov testera';
			SC_P3_HV_Test.IdleTime.PT:= T#1s;
			SC_P3_HV_Test.AlarmTime.PT:= T#5s;

			P3_HV_Test.OUT.PritlacenieKontaktovTestera_ON:= TRUE;
			SC_P3_HV_Test.IdleTime.IN:= TRUE;

			IF SC_P3_HV_Test.IdleTime.Q THEN
				IF P3_HV_Test.Manual THEN
					IF NOT P3_HV_Test.CMD.RR_ZatvorTester THEN
						SC_P3_HV_Test.ResetStep:= TRUE;
						SC_P3_HV_Test.Step:= 140;
					END_IF
				ELSE
					SC_P3_HV_Test.ResetStep:= TRUE;
					SC_P3_HV_Test.Step:= 130;
				END_IF
			END_IF

		130:
			SC_P3_HV_Test.StepName:='130 - Automaticky Rezim - spustenie testera';
			SC_P3_HV_Test.IdleTime.PT:= T#2s;
			SC_P3_HV_Test.AlarmTime.PT:= T#5s;

			SC_P3_HV_Test.IdleTime.IN:= TRUE;
			IF Linka.KOM_Panatrace_OFF THEN
				IF SC_P3_HV_Test.IdleTime.Q THEN
					SC_P3_HV_Test.ResetStep:= TRUE;
					SC_P3_HV_Test.Step:= 140;
				END_IF
			ELSE
				P3_HV_Test.STAV.Vysledok_HV_Testu:= '';
				P3_HV_Test.CMD.StartTestovania:= TRUE;
				P3_HVtest_Taktime.IN.START_MeraniaStratovehoCasu:= TRUE;
				SC_P3_HV_Test.ResetStep:= TRUE;
				SC_P3_HV_Test.Step:= 133;
			END_IF

		133:
			SC_P3_HV_Test.StepName:='133 - Automaticky Rezim - cakam na ukoncenie HV testu';
			SC_P3_HV_Test.IdleTime.PT:= T#1s;
			SC_P3_HV_Test.AlarmTime.PT:= T#5s;

			IF P3_HV_Test.STAV.TestovanieUkoncene THEN
				P3_HVtest_Taktime.IN.START_MeraniaStratovehoCasu:= FALSE;
				Paletka[i].STAV.HV_Test_Ukonceny:= TRUE;
				P3_HV_Test.CMD.StartTestovania:= FALSE;
				IF Paletka[i].STAV.StavPaletky = 'TEST' THEN
					SC_P3_HV_Test.ResetStep:= TRUE;
					SC_P3_HV_Test.Step:= 135;
				ELSE
					IF P3_HV_Test.STAV.Vysledok_HV_Testu = 'OK' THEN
						Paletka[i].STAV.StavPaletky:= 'OK';
					ELSIF P3_HV_Test.STAV.Vysledok_HV_Testu = 'NG' THEN
						Paletka[i].STAV.StavPaletky:= 'NG';
					END_IF
					SC_P3_HV_Test.ResetStep:= TRUE;
					SC_P3_HV_Test.Step:= 135;
				END_IF
			ELSIF P3_HV_Test.STAV.TesterNeodpoveda THEN
				P3_HV_Test.CMD.StartTestovania:= FALSE;
				SC_P3_HV_Test.ResetStep:= TRUE;
				SC_P3_HV_Test.Step:= 134;
			END_IF

		134:
			SC_P3_HV_Test.StepName:='134 - Automaticky Rezim - zobrazenie hlasenia tester neodpoveda';
			SC_P3_HV_Test.IdleTime.PT:= T#1s;
			SC_P3_HV_Test.AlarmTime.PT:= T#5s;

			P34_Vizu.ZobrazHL1_HVtest:= TRUE;

			IF P3_HV_Test.CMD.OpatovnyTest THEN
				P3_HV_Test.CMD.OpatovnyTest:= FALSE;
				P34_Vizu.ZobrazHL1_HVtest:= FALSE;
				IF P3_HV_Test.PAR.CisloPortuKlienta < 1039 THEN
					P3_HV_Test.PAR.CisloPortuKlienta:= P3_HV_Test.PAR.CisloPortuKlienta + 1;
				ELSE
					P3_HV_Test.PAR.CisloPortuKlienta:= 1031;
				END_IF
				SC_P3_HV_Test.ResetStep:= TRUE;
				SC_P3_HV_Test.Step:= 130;
			ELSIF P3_HV_Test.STAV.PaletkaOznacena_NG THEN
				P3_HV_Test.STAV.PaletkaOznacena_NG:= FALSE;
				P34_Vizu.ZobrazHL1_HVtest:= FALSE;
				Paletka[i].STAV.StavPaletky:= 'NG';
				SC_P3_HV_Test.ResetStep:= TRUE;
				SC_P3_HV_Test.Step:= 135;
			END_IF

		135:
			SC_P3_HV_Test.StepName:='135 - Automaticky Rezim - cakam na zrusenie signalu HV test ukonceny';
			SC_P3_HV_Test.IdleTime.PT:= T#1s;
			SC_P3_HV_Test.AlarmTime.PT:= T#5s;

			IF NOT P3_HV_Test.STAV.TestovanieUkoncene THEN
				SC_P3_HV_Test.ResetStep:= TRUE;
				SC_P3_HV_Test.Step:= 140;
			END_IF

			//Otvorenie HV testera//

		140:
			SC_P3_HV_Test.StepName:='140 - Automaticky Rezim - zasunutie pritlacenia kontaktov testera';
			SC_P3_HV_Test.IdleTime.PT:= T#1s;
			SC_P3_HV_Test.AlarmTime.PT:= T#5s;

			P3_HV_Test.OUT.PritlacenieKontaktovTestera_ON:= FALSE;
			SC_P3_HV_Test.IdleTime.IN:= TRUE;

			IF SC_P3_HV_Test.IdleTime.Q THEN
				SC_P3_HV_Test.ResetStep:= TRUE;
				SC_P3_HV_Test.Step:= 143;
			END_IF

		143:
			SC_P3_HV_Test.StepName:='143 - Automaticky Rezim - zasunutie spodnych kontaktov';
			SC_P3_HV_Test.IdleTime.PT:= T#200ms;
			SC_P3_HV_Test.AlarmTime.PT:= T#5s;

			IF NOT SC_P3_HV_Test.Switch1 THEN
				SpodneKontakty_ZASUN:= TRUE;
				SC_P3_HV_Test.Switch1:= TRUE;
			END_IF

			IF P3_HV_Test.IN.SpodneKontakty_ZASUNUTE THEN
				SC_P3_HV_Test.ResetStep:= TRUE;
				SC_P3_HV_Test.Step:= 145;
			END_IF

		145:
			SC_P3_HV_Test.StepName:='145 - Automaticky Rezim - zasunutie hornych kontaktov';
			SC_P3_HV_Test.IdleTime.PT:= T#200ms;
			SC_P3_HV_Test.AlarmTime.PT:= T#5s;

			IF NOT SC_P3_HV_Test.Switch1 THEN
				HorneKontakty_ZASUN:= TRUE;
				SC_P3_HV_Test.Switch1:= TRUE;
			END_IF

			IF P3_HV_Test.IN.HorneKontakty_ZASUNUTE THEN
				SC_P3_HV_Test.ResetStep:= TRUE;
				SC_P3_HV_Test.Step:= 148;
			END_IF

		148:
			SC_P3_HV_Test.StepName:='148 - Automaticky Rezim - zasunutie pruzenia hornych kontaktov';
			SC_P3_HV_Test.IdleTime.PT:= T#500ms;
			SC_P3_HV_Test.AlarmTime.PT:= T#5s;

			IF NOT SC_P3_HV_Test.Switch1 THEN
				P3_HV_Test.OUT.PruzenieHornychKontaktov_VYSUN:= FALSE;
				P3_HV_Test.OUT.PruzenieHornychKontaktov_ZASUN:= TRUE;
				SC_P3_HV_Test.IdleTime.IN:= TRUE;
			END_IF

			IF SC_P3_HV_Test.IdleTime.Q THEN
				SC_P3_HV_Test.ResetStep:= TRUE;
				SC_P3_HV_Test.Step:= 150;
			END_IF

		150:
			SC_P3_HV_Test.StepName:='150 - Automaticky Rezim - odcentrovanie paletky';
			SC_P3_HV_Test.IdleTime.PT:= T#200ms;
			SC_P3_HV_Test.AlarmTime.PT:= T#5s;

			IF NOT SC_P3_HV_Test.Switch1 THEN
				Centrovacku_ZASUN:= TRUE;
				SC_P3_HV_Test.Switch1:= TRUE;
			END_IF

			IF P3_HV_Test.IN.Centrovanie_ZASUNUTE THEN
				IF P3_HV_Test.Manual THEN
					P3_HV_Test.STAV.RR_SekvenciaTestera_BUSY:= FALSE;
					SC_P3_HV_Test.ResetStep:= TRUE;
					SC_P3_HV_Test.Step:= 700;
				ELSE
					SC_P3_HV_Test.ResetStep:= TRUE;
					SC_P3_HV_Test.Step:= 560;
				END_IF
			END_IF

			//***************************Vyvezenie paletky**********************************************//
		560:
			SC_P3_HV_Test.StepName:='560 - Automaticky Rezim - cakam na vyvezenie na zdvižku pred Leakage Testom A';
			SC_P3_HV_Test.IdleTime.PT:= T#200ms;
			SC_P3_HV_Test.AlarmTime.PT:= T#5s;

			IF P3_HV_Test.KoniecCyklu THEN
				SC_P3_HV_Test.ResetStep:= TRUE;
				SC_P3_HV_Test.Step:= 0;
			ELSIF NOT P3_ZdvizkaPredLeakTestA.IN.PritomnostPaletky AND
				SC_P3_ZdvizkaPredLeakTestA.Step = 100 AND
				NOT P3_HV_Test.STAV.PrebiehaVyvezeniePaletky AND
				P3_ZdvizkaPredLeakTestA.STAV.PoINIT THEN
				P3_HV_Test.OUT.ZasunStoper:= TRUE;
				P3_HV_Test.STAV.PrebiehaVyvezeniePaletky:= TRUE;
				SC_P3_HV_Test.ResetStep:= TRUE;
				SC_P3_HV_Test.Step:= 561;
			END_IF

		561:
			SC_P3_HV_Test.StepName:='561 - Automaticky Rezim - ukoncenie vyvazania na zdvižku pred Leakage Testom A';
			SC_P3_HV_Test.IdleTime.PT:= T#200ms;
			SC_P3_HV_Test.AlarmTime.PT:= T#10s;

			SC_P3_HV_Test.AlarmTime.IN:= P3_HV_Test.RFID_hlava.PritomnostPaletky;
			SC_P3_HV_Test.IdleTime.IN:= NOT P3_HV_Test.RFID_hlava.PritomnostPaletky;

			IF NOT P3_HV_Test.RFID_hlava.PritomnostPaletky THEN
				TestovaciKus:= FALSE;
				Paletka[i].PAR.StavPowerCP:= '';
				Paletka[i].STAV.Komunikacia_DONE:= FALSE;
				Paletka[i].STAV.OdoslanieFotiek_DONE:= FALSE;
				P3_HV_Test.OUT.ZasunStoper:= FALSE;
				SC_P3_HV_Test.ResetStep:= TRUE;
				SC_P3_HV_Test.Step:= 100;
			ELSIF SC_P3_HV_Test.AlarmTime.Q THEN
				P34_Alarmy[367]:= TRUE;
				P3_Pracovisko.STAV.Porucha_ST2:= TRUE;
			END_IF

			//*******************************************************Manuálny režim*******************************************************************************//

		700:
			SC_P3_HV_Test.StepName:='700 - Manualny Rezim';
			SC_P3_HV_Test.IdleTime.PT:= T#8s;
			SC_P3_HV_Test.AlarmTime.PT:= T#5s;

			//Sekvencia zatvorenia testera//
			IF P3_HV_Test.CMD.RR_ZatvorTester THEN
				P3_HV_Test.STAV.RR_SekvenciaTestera_BUSY:= TRUE;
				SC_P3_HV_Test.ResetStep:= TRUE;
				SC_P3_HV_Test.Step:= 110;
			END_IF

			//Ovládanie zdvižky//
			IF P3_HV_Test.CMD.RR_VysunCentrovanie THEN
				P3_HV_Test.OUT.Centrovanie_VYSUN:= TRUE;
				P3_HV_Test.OUT.Centrovanie_ZASUN:= FALSE;
			ELSE
				P3_HV_Test.OUT.Centrovanie_VYSUN:= FALSE;
				P3_HV_Test.OUT.Centrovanie_ZASUN:= TRUE;
			END_IF

			//Ovládanie pruženia horných kontaktov//
			IF P3_HV_Test.CMD.RR_VysunPruzenieKontaktov THEN
				P3_HV_Test.OUT.PruzenieHornychKontaktov_ZASUN:= FALSE;
				P3_HV_Test.OUT.PruzenieHornychKontaktov_VYSUN:= TRUE;
			ELSE
				P3_HV_Test.OUT.PruzenieHornychKontaktov_ZASUN:= TRUE;
				P3_HV_Test.OUT.PruzenieHornychKontaktov_VYSUN:= FALSE;
			END_IF

	END_CASE

END_PROGRAM

PROGRAM _EXIT
	(* Insert code here *)

END_PROGRAM
```

#### Variables.var - Local variables
```iecst
VAR
	SC_OvlCentrovacky : SequenceControlTyp;
	Centrovacku_VYSUN : BOOL;
	Centrovacku_ZASUN : BOOL;
	SC_OvlSpodnychKontaktov : SequenceControlTyp;
	SpodneKontakty_VYSUN : BOOL;
	SpodneKontakty_ZASUN : BOOL;
	SC_OvlHornychKontaktov : SequenceControlTyp;
	HorneKontakty_VYSUN : BOOL;
	HorneKontakty_ZASUN : BOOL;
	i : USINT;
	TestovaciKus : BOOL := 0;
	SC_OvlTesteraHV : SequenceControlTyp;
	SKTcpClientTester_0 : SKTcpClientTester;
	dataStr : STRING[32];
	PocetDopytovNaTester : USINT;
	Cas_HVTester : TON;
END_VAR
```

#### IOLinkKomunikacia.st
```iecst
ACTION IOLinkKomunikacia:

	//RFID snímač paletky//
	P3_HV_Test.RFID_hlava();

END_ACTION
```

#### OvlCentrovacky.st
```iecst
ACTION OvlCentrovacky:

	//Volanie funkcie SequenceControl//
	SequenceControl(SC:= SC_OvlCentrovacky);

	CASE SC_OvlCentrovacky.Step OF

		0:
			SC_OvlCentrovacky.StepName:= '0 - Nulovanie';
			Centrovacku_VYSUN:= FALSE;
			Centrovacku_ZASUN:= FALSE;

			IF SC_P3_HV_Test.Step <> 0 THEN
				SC_OvlCentrovacky.ResetStep:= TRUE;
				SC_OvlCentrovacky.Step:= 1;
			END_IF

		1:
			SC_OvlCentrovacky.StepName:= '1 - Rozhodnutie o cinnosti';
			IF Centrovacku_VYSUN THEN
				SC_OvlCentrovacky.Step:= 10;
			ELSIF Centrovacku_ZASUN THEN
				SC_OvlCentrovacky.Step:= 20;
			END_IF

		10:
			SC_OvlCentrovacky.StepName:= '10 - Vysunutie centrovacky';
			SC_OvlCentrovacky.IdleTime.PT:= T#3s;
			SC_OvlCentrovacky.AlarmTime.PT:= T#6s;

			IF P3_HV_Test.Automat THEN
				SC_OvlCentrovacky.AlarmTime.IN:= TRUE;
			ELSE
				SC_OvlCentrovacky.IdleTime.IN:= TRUE;
			END_IF

			IF NOT SC_OvlCentrovacky.Switch1 THEN
				P3_HV_Test.OUT.Centrovanie_ZASUN:= FALSE;
                P3_HV_Test.OUT.Centrovanie_VYSUN:= TRUE;
				SC_OvlCentrovacky.Switch1:= TRUE;
			END_IF

			IF P3_HV_Test.IN.Centrovanie_VYSUNUTE OR SC_OvlCentrovacky.IdleTime.Q THEN
				SC_OvlCentrovacky.ResetStep:= TRUE;
				SC_OvlCentrovacky.Step:= 0;
			ELSIF SC_OvlCentrovacky.AlarmTime.Q THEN
				P34_Alarmy[360]:= TRUE;
				P3_Pracovisko.STAV.Porucha_ST2:= TRUE;
			END_IF

		20:
			SC_OvlCentrovacky.StepName:= '20 - Zasunutie centrovacky';
			SC_OvlCentrovacky.IdleTime.PT:= T#3s;
			SC_OvlCentrovacky.AlarmTime.PT:= T#6s;

			IF P3_HV_Test.Automat THEN
				SC_OvlCentrovacky.AlarmTime.IN:= TRUE;
			ELSE
				SC_OvlCentrovacky.IdleTime.IN:= TRUE;
			END_IF

			IF NOT SC_OvlCentrovacky.Switch1 THEN
				P3_HV_Test.OUT.Centrovanie_VYSUN:= FALSE;
                P3_HV_Test.OUT.Centrovanie_ZASUN:= TRUE;
				SC_OvlCentrovacky.Switch1:= TRUE;
			END_IF

			IF P3_HV_Test.IN.Centrovanie_ZASUNUTE OR SC_OvlCentrovacky.IdleTime.Q THEN
				SC_OvlCentrovacky.ResetStep:= TRUE;
				SC_OvlCentrovacky.Step:= 0;
			ELSIF SC_OvlCentrovacky.AlarmTime.Q THEN
				P34_Alarmy[361]:= TRUE;
				P3_Pracovisko.STAV.Porucha_ST2:= TRUE;
			END_IF

	END_CASE

END_ACTION
```

#### OvlSpodnychKontaktov.st
```iecst
ACTION OvlSpodnychKontaktov:

	//Volanie funkcie SequenceControl//
	SequenceControl(SC:= SC_OvlSpodnychKontaktov);

	CASE SC_OvlSpodnychKontaktov.Step OF

		0:
			SC_OvlSpodnychKontaktov.StepName:= '0 - Nulovanie';
			SpodneKontakty_VYSUN:= FALSE;
			SpodneKontakty_ZASUN:= FALSE;

			IF SC_P3_HV_Test.Step <> 0 THEN
				SC_OvlSpodnychKontaktov.ResetStep:= TRUE;
				SC_OvlSpodnychKontaktov.Step:= 1;
			END_IF

		1:
			SC_OvlSpodnychKontaktov.StepName:= '1 - Rozhodnutie o cinnosti';
			IF SpodneKontakty_VYSUN THEN
				SC_OvlSpodnychKontaktov.Step:= 10;
			ELSIF SpodneKontakty_ZASUN THEN
				SC_OvlSpodnychKontaktov.Step:= 20;
			END_IF

		10:
			SC_OvlSpodnychKontaktov.StepName:= '10 - Vysunutie spodnych kontaktov';
			SC_OvlSpodnychKontaktov.IdleTime.PT:= T#3s;
			SC_OvlSpodnychKontaktov.AlarmTime.PT:= T#6s;

			IF P3_HV_Test.Automat THEN
				SC_OvlSpodnychKontaktov.AlarmTime.IN:= TRUE;
			ELSE
				SC_OvlSpodnychKontaktov.IdleTime.IN:= TRUE;
			END_IF

			IF NOT SC_OvlSpodnychKontaktov.Switch1 THEN
				P3_HV_Test.OUT.SpodneKontakty_ZASUN:= FALSE;
                P3_HV_Test.OUT.SpodneKontakty_VYSUN:= TRUE;
				SC_OvlSpodnychKontaktov.Switch1:= TRUE;
			END_IF

			IF P3_HV_Test.IN.SpodneKontakty_VYSUNUTE OR SC_OvlSpodnychKontaktov.IdleTime.Q THEN
				SC_OvlSpodnychKontaktov.ResetStep:= TRUE;
				SC_OvlSpodnychKontaktov.Step:= 0;
			ELSIF SC_OvlSpodnychKontaktov.AlarmTime.Q THEN
				P34_Alarmy[362]:= TRUE;
				P3_Pracovisko.STAV.Porucha_ST2:= TRUE;
			END_IF

		20:
			SC_OvlSpodnychKontaktov.StepName:= '20 - Zasunutie spodnych kontaktov';
			SC_OvlSpodnychKontaktov.IdleTime.PT:= T#3s;
			SC_OvlSpodnychKontaktov.AlarmTime.PT:= T#6s;

			IF P3_HV_Test.Automat THEN
				SC_OvlSpodnychKontaktov.AlarmTime.IN:= TRUE;
			ELSE
				SC_OvlSpodnychKontaktov.IdleTime.IN:= TRUE;
			END_IF

			IF NOT SC_OvlSpodnychKontaktov.Switch1 THEN
				P3_HV_Test.OUT.SpodneKontakty_VYSUN:= FALSE;
                P3_HV_Test.OUT.SpodneKontakty_ZASUN:= TRUE;
				SC_OvlSpodnychKontaktov.Switch1:= TRUE;
			END_IF

			IF P3_HV_Test.IN.SpodneKontakty_ZASUNUTE OR SC_OvlSpodnychKontaktov.IdleTime.Q THEN
				SC_OvlSpodnychKontaktov.ResetStep:= TRUE;
				SC_OvlSpodnychKontaktov.Step:= 0;
			ELSIF SC_OvlSpodnychKontaktov.AlarmTime.Q THEN
				P34_Alarmy[363]:= TRUE;
				P3_Pracovisko.STAV.Porucha_ST2:= TRUE;
			END_IF

	END_CASE

END_ACTION
```

#### OvlHornychKontaktov.st
```iecst
ACTION OvlHornychKontaktov:

	//Volanie funkcie SequenceControl//
	SequenceControl(SC:= SC_OvlHornychKontaktov);

	CASE SC_OvlHornychKontaktov.Step OF

		0:
			SC_OvlHornychKontaktov.StepName:= '0 - Nulovanie';
			HorneKontakty_VYSUN:= FALSE;
			HorneKontakty_ZASUN:= FALSE;

			IF SC_P3_HV_Test.Step <> 0 THEN
				SC_OvlHornychKontaktov.ResetStep:= TRUE;
				SC_OvlHornychKontaktov.Step:= 1;
			END_IF

		1:
			SC_OvlHornychKontaktov.StepName:= '1 - Rozhodnutie o cinnosti';
			IF HorneKontakty_VYSUN THEN
				SC_OvlHornychKontaktov.Step:= 10;
			ELSIF HorneKontakty_ZASUN THEN
				SC_OvlHornychKontaktov.Step:= 20;
			END_IF

		10:
			SC_OvlHornychKontaktov.StepName:= '10 - Vysunutie hornych kontaktov';
			SC_OvlHornychKontaktov.IdleTime.PT:= T#3s;
			SC_OvlHornychKontaktov.AlarmTime.PT:= T#6s;

			IF P3_HV_Test.Automat THEN
				SC_OvlHornychKontaktov.AlarmTime.IN:= TRUE;
			ELSE
				SC_OvlHornychKontaktov.IdleTime.IN:= TRUE;
			END_IF

			IF NOT SC_OvlHornychKontaktov.Switch1 THEN
				P3_HV_Test.OUT.HorneKontakty_ZASUN:= FALSE;
				P3_HV_Test.OUT.HorneKontakty_VYSUN:= TRUE;
				SC_OvlHornychKontaktov.Switch1:= TRUE;
			END_IF

			IF P3_HV_Test.IN.HorneKontakty_VYSUNUTE OR SC_OvlHornychKontaktov.IdleTime.Q THEN
				SC_OvlHornychKontaktov.ResetStep:= TRUE;
				SC_OvlHornychKontaktov.Step:= 0;
			ELSIF SC_OvlHornychKontaktov.AlarmTime.Q THEN
				P34_Alarmy[364]:= TRUE;
				P3_Pracovisko.STAV.Porucha_ST2:= TRUE;
			END_IF

		20:
			SC_OvlHornychKontaktov.StepName:= '20 - Zasunutie hornych kontaktov';
			SC_OvlHornychKontaktov.IdleTime.PT:= T#3s;
			SC_OvlHornychKontaktov.AlarmTime.PT:= T#6s;

			IF P3_HV_Test.Automat THEN
				SC_OvlHornychKontaktov.AlarmTime.IN:= TRUE;
			ELSE
				SC_OvlHornychKontaktov.IdleTime.IN:= TRUE;
			END_IF

			IF NOT SC_OvlHornychKontaktov.Switch1 THEN
				P3_HV_Test.OUT.HorneKontakty_VYSUN:= FALSE;
				P3_HV_Test.OUT.HorneKontakty_ZASUN:= TRUE;
				SC_OvlHornychKontaktov.Switch1:= TRUE;
			END_IF

			IF P3_HV_Test.IN.HorneKontakty_ZASUNUTE OR SC_OvlHornychKontaktov.IdleTime.Q THEN
				SC_OvlHornychKontaktov.ResetStep:= TRUE;
				SC_OvlHornychKontaktov.Step:= 0;
			ELSIF SC_OvlHornychKontaktov.AlarmTime.Q THEN
				P34_Alarmy[365]:= TRUE;
				P3_Pracovisko.STAV.Porucha_ST2:= TRUE;
			END_IF

	END_CASE

END_ACTION
```

#### COM_Tester.st
```iecst
ACTION COM_Tester:

	//Parametre komunikácie//
    memcpy(ADR(SKTcpClientTester_0.Params.IPaddrServ),ADR('192.168.128.251'),SIZEOF('192.168.128.251'));
    SKTcpClientTester_0.Params.IPportClient := P3_HV_Test.PAR.CisloPortuKlienta;
    SKTcpClientTester_0.Params.IPportServ := 1030;
    SKTcpClientTester_0.Params.RecvTimeout := 10000;
    strcpy(ADR(SKTcpClientTester_0.Params.Packet.data),ADR(dataStr));
    SKTcpClientTester_0();

    Cas_HVTester.PT:= T#1M;
    Cas_HVTester();

    //Volanie funkcie SequenceControl//
    SequenceControl(SC:= SC_OvlTesteraHV);

    CASE SC_OvlTesteraHV.Step OF

        0:
            SC_OvlTesteraHV.StepName:= '0 - Nulovanie';
            SKTcpClientTester_0.Enable:= TRUE;
            SKTcpClientTester_0.Cmd.Send:= FALSE;
			P3_HV_Test.STAV.TestovanieUkoncene:= FALSE;
			P3_HV_Test.STAV.TesterNeodpoveda:= FALSE;
            PocetDopytovNaTester:= 0;
            SC_OvlTesteraHV.ResetStep:= TRUE;
            SC_OvlTesteraHV.Step:= 1;

        1:
            SC_OvlTesteraHV.StepName:= '1 - Cakam na spustenie testera';
            IF P3_HV_Test.CMD.StartTestovania THEN
                P3_HV_Test.STAV.Vysledok_HV_Testu:= '';
                Cas_HVTester.IN:= TRUE;
                P3_HV_Test.STAV.NameranyCas_InitTestera:= 0;
                P3_HV_Test.STAV.NameranyCas_PoslanieQRkodu:= 0;
                P3_HV_Test.STAV.NameranyCas_CelkovyCasTestovania:= 0;
                SC_OvlTesteraHV.Step:= 10;
            END_IF

        10:
            SC_OvlTesteraHV.StepName:= '10 - Dopyt na stav testera - typ 0';
            SC_OvlTesteraHV.IdleTime.PT:= T#300ms;
            SC_OvlTesteraHV.AlarmTime.PT:= T#5s;
            SC_OvlTesteraHV.IdleTime.IN:= TRUE;
            SC_OvlTesteraHV.AlarmTime.IN:= TRUE;

            SKTcpClientTester_0.Params.Packet.type:= 0;
            SKTcpClientTester_0.Params.Packet.workplace:= 46;
            SKTcpClientTester_0.Params.Packet.id:= 1;
            SKTcpClientTester_0.Cmd.Close:= FALSE;
			SKTcpClientTester_0.Cmd.Send:= TRUE;

            IF SKTcpClientTester_0.Cmd.Send AND NOT SKTcpClientTester_0.Status.staReceived AND NOT SKTcpClientTester_0.Status.staError THEN
                SC_OvlTesteraHV.ResetStep:= TRUE;
                SC_OvlTesteraHV.Step:= 13;
            ELSIF SC_OvlTesteraHV.AlarmTime.Q AND (SKTcpClientTester_0.Status.staReceived OR SKTcpClientTester_0.Status.staError) THEN
                PocetDopytovNaTester:= PocetDopytovNaTester + 1;
				SKTcpClientTester_0.Cmd.Send:= FALSE;
				SKTcpClientTester_0.Cmd.Close:= TRUE;
				SC_OvlTesteraHV.ResetStep:= TRUE;
                SC_OvlTesteraHV.Step:= 12;
            END_IF

        12:
            SC_OvlTesteraHV.StepName:= '12 - Dopyt na stav testera - cakam na opatovny dopyt na tester';
            SC_OvlTesteraHV.IdleTime.PT:= T#800ms;
            SC_OvlTesteraHV.AlarmTime.PT:= T#5s;
            SC_OvlTesteraHV.IdleTime.IN:= TRUE;
            SKTcpClientTester_0.Cmd.Send:= FALSE;

            IF PocetDopytovNaTester < 3 THEN
                IF SC_OvlTesteraHV.IdleTime.Q THEN
                    SC_OvlTesteraHV.ResetStep:= TRUE;
                    SC_OvlTesteraHV.Step:= 10;
                END_IF
            ELSE
                P3_HV_Test.STAV.Vysledok_HV_Testu:= 'NG';
                P3_HV_Test.STAV.TesterNeodpoveda:= TRUE;
                SC_OvlTesteraHV.ResetStep:= TRUE;
                SC_OvlTesteraHV.Step:= 100;
            END_IF

        13:
            SC_OvlTesteraHV.StepName:= '13 - Odpoved na stav testera - typ 0';
            SC_OvlTesteraHV.IdleTime.PT:= T#800ms;
            SC_OvlTesteraHV.AlarmTime.PT:= T#10s;
            SC_OvlTesteraHV.IdleTime.IN:= TRUE;

            IF SKTcpClientTester_0.Status.staReceived AND SKTcpClientTester_0.Status.DataRecv[2]= 0 AND SKTcpClientTester_0.Status.DataRecv[5]= 2 THEN
                SKTcpClientTester_0.Cmd.Send:= FALSE;
                P3_HV_Test.STAV.NameranyCas_InitTestera:= Cas_HVTester.ET;
                SC_OvlTesteraHV.ResetStep:= TRUE;
                SC_OvlTesteraHV.Step:= 15;
            ELSIF SKTcpClientTester_0.Status.staReceived AND SKTcpClientTester_0.Status.DataRecv[2]= 0 AND SKTcpClientTester_0.Status.DataRecv[5]= 1 THEN
                SKTcpClientTester_0.Cmd.Send:= FALSE;
                SKTcpClientTester_0.Cmd.Close:= TRUE;
				IF SC_OvlTesteraHV.IdleTime.Q THEN
                    SC_OvlTesteraHV.ResetStep:= TRUE;
                    SC_OvlTesteraHV.Step:= 10;
                END_IF
            ELSIF SKTcpClientTester_0.Status.staReceived AND SKTcpClientTester_0.Status.DataRecv[2]= 0 AND SKTcpClientTester_0.Status.DataRecv[5]= 0 THEN
                SKTcpClientTester_0.Cmd.Send:= FALSE;
                SKTcpClientTester_0.Cmd.Close:= TRUE;
				IF SC_OvlTesteraHV.IdleTime.Q THEN
                    SC_OvlTesteraHV.ResetStep:= TRUE;
                    SC_OvlTesteraHV.Step:= 10;
                END_IF
            ELSIF SKTcpClientTester_0.Status.staError THEN
                SKTcpClientTester_0.Cmd.Send:= FALSE;
                P3_HV_Test.STAV.Vysledok_HV_Testu:= 'NG';
                P3_HV_Test.STAV.TesterNeodpoveda:= TRUE;
                SC_OvlTesteraHV.ResetStep:= TRUE;
                SC_OvlTesteraHV.Step:= 100;
            END_IF

        15:
            SC_OvlTesteraHV.StepName:= '15 - Poslanie QR kodu Power CP - typ 1';
            SC_OvlTesteraHV.IdleTime.PT:= T#300ms;
            SC_OvlTesteraHV.AlarmTime.PT:= T#10s;
            SC_OvlTesteraHV.IdleTime.IN:= TRUE;

            SKTcpClientTester_0.Params.Packet.type:= 1;
            SKTcpClientTester_0.Params.Packet.workplace:= 46;
            SKTcpClientTester_0.Params.Packet.id:= 1;
			dataStr:= Paletka[i].PAR.QRkodPowerCP;
	        SKTcpClientTester_0.Cmd.Send:= TRUE;

            IF SKTcpClientTester_0.Cmd.Send AND NOT SKTcpClientTester_0.Status.staReceived AND NOT SKTcpClientTester_0.Status.staError THEN
                SC_OvlTesteraHV.ResetStep:= TRUE;
                SC_OvlTesteraHV.Step:= 18;
            END_IF

        18:
            SC_OvlTesteraHV.StepName:= '18 - Odpoved na poslanie QR kodu - typ 1';
            SC_OvlTesteraHV.IdleTime.PT:= T#300ms;
            SC_OvlTesteraHV.AlarmTime.PT:= T#10s;
            SC_OvlTesteraHV.IdleTime.IN:= TRUE;

            IF SKTcpClientTester_0.Status.staReceived AND SKTcpClientTester_0.Status.DataRecv[2]= 1 AND SKTcpClientTester_0.Status.DataRecv[5]= 0 THEN
                SKTcpClientTester_0.Cmd.Send:= FALSE;
                P3_HV_Test.STAV.NameranyCas_PoslanieQRkodu:= Cas_HVTester.ET;
                SC_OvlTesteraHV.ResetStep:= TRUE;
                SC_OvlTesteraHV.Step:= 20;
            ELSIF SKTcpClientTester_0.Status.staReceived AND SKTcpClientTester_0.Status.DataRecv[2]= 1 AND SKTcpClientTester_0.Status.DataRecv[5]= 2 THEN
                SKTcpClientTester_0.Cmd.Send:= FALSE;
                IF SC_OvlTesteraHV.IdleTime.Q THEN
                    SC_OvlTesteraHV.ResetStep:= TRUE;
                    SC_OvlTesteraHV.Step:= 15;
                END_IF
            ELSIF SKTcpClientTester_0.Status.staReceived AND SKTcpClientTester_0.Status.DataRecv[2]= 1 AND SKTcpClientTester_0.Status.DataRecv[5]= 1 THEN
                SKTcpClientTester_0.Cmd.Send:= FALSE;
                P3_HV_Test.STAV.Vysledok_HV_Testu:= 'NG';
                P3_HV_Test.STAV.TestovanieUkoncene:= TRUE;
                SC_OvlTesteraHV.ResetStep:= TRUE;
                SC_OvlTesteraHV.Step:= 100;
            ELSIF SKTcpClientTester_0.Status.staError THEN
                SKTcpClientTester_0.Cmd.Send:= FALSE;
                P3_HV_Test.STAV.Vysledok_HV_Testu:= 'NG';
                P3_HV_Test.STAV.TesterNeodpoveda:= TRUE;
                SC_OvlTesteraHV.ResetStep:= TRUE;
                SC_OvlTesteraHV.Step:= 100;
            END_IF

        20:
            SC_OvlTesteraHV.StepName:= '20 - Dopyt na stav testera - typ 0';
            SC_OvlTesteraHV.IdleTime.PT:= T#300ms;
            SC_OvlTesteraHV.AlarmTime.PT:= T#10s;
            SC_OvlTesteraHV.IdleTime.IN:= TRUE;

            SKTcpClientTester_0.Params.Packet.type:= 0;
            SKTcpClientTester_0.Params.Packet.workplace:= 46;
            SKTcpClientTester_0.Params.Packet.id:= 1;
            SKTcpClientTester_0.Cmd.Send:= TRUE;

            IF SKTcpClientTester_0.Cmd.Send AND NOT SKTcpClientTester_0.Status.staReceived AND NOT SKTcpClientTester_0.Status.staError THEN
                SC_OvlTesteraHV.ResetStep:= TRUE;
                SC_OvlTesteraHV.Step:= 23;
            END_IF

        23:
            SC_OvlTesteraHV.StepName:= '23 - Odpoved na stav testera - typ 0';
            SC_OvlTesteraHV.IdleTime.PT:= T#300ms;
            SC_OvlTesteraHV.AlarmTime.PT:= T#10s;
            SC_OvlTesteraHV.IdleTime.IN:= TRUE;

            IF SKTcpClientTester_0.Status.staReceived AND SKTcpClientTester_0.Status.DataRecv[2]= 0 AND SKTcpClientTester_0.Status.DataRecv[5]= 3 THEN
                SKTcpClientTester_0.Cmd.Send:= FALSE;
                IF SC_OvlTesteraHV.IdleTime.Q THEN
                    SC_OvlTesteraHV.ResetStep:= TRUE;
                    SC_OvlTesteraHV.Step:= 20;
                END_IF
            ELSIF SKTcpClientTester_0.Status.staReceived AND SKTcpClientTester_0.Status.DataRecv[2]= 0 AND SKTcpClientTester_0.Status.DataRecv[5]= 4 THEN
                SKTcpClientTester_0.Cmd.Send:= FALSE;
                SC_OvlTesteraHV.ResetStep:= TRUE;
                SC_OvlTesteraHV.Step:= 25;
            ELSIF SKTcpClientTester_0.Status.staReceived AND SKTcpClientTester_0.Status.DataRecv[2]= 0 AND SKTcpClientTester_0.Status.DataRecv[5]= 0 THEN
                SKTcpClientTester_0.Cmd.Send:= FALSE;
                P3_HV_Test.STAV.Vysledok_HV_Testu:= 'NG';
                P3_HV_Test.STAV.TestovanieUkoncene:= TRUE;
                SC_OvlTesteraHV.ResetStep:= TRUE;
                SC_OvlTesteraHV.Step:= 100;
            ELSIF SKTcpClientTester_0.Status.staError THEN
                SKTcpClientTester_0.Cmd.Send:= FALSE;
                P3_HV_Test.STAV.Vysledok_HV_Testu:= 'NG';
                P3_HV_Test.STAV.TesterNeodpoveda:= TRUE;
                SC_OvlTesteraHV.ResetStep:= TRUE;
                SC_OvlTesteraHV.Step:= 100;
            END_IF

        25:
            SC_OvlTesteraHV.StepName:= '25 - Dopyt na vysledok testu - typ 2';
            SC_OvlTesteraHV.IdleTime.PT:= T#300ms;
            SC_OvlTesteraHV.AlarmTime.PT:= T#10s;
            SC_OvlTesteraHV.IdleTime.IN:= TRUE;

            SKTcpClientTester_0.Params.Packet.type:= 2;
            SKTcpClientTester_0.Params.Packet.workplace:= 46;
            SKTcpClientTester_0.Params.Packet.id:= 1;
            SKTcpClientTester_0.Cmd.Send:= TRUE;

            IF SKTcpClientTester_0.Cmd.Send AND NOT SKTcpClientTester_0.Status.staReceived AND NOT SKTcpClientTester_0.Status.staError THEN
                SC_OvlTesteraHV.ResetStep:= TRUE;
                SC_OvlTesteraHV.Step:= 28;
            END_IF

        28:
            SC_OvlTesteraHV.StepName:= '28 - Odpoved na vysledok testu - typ 2';
            SC_OvlTesteraHV.IdleTime.PT:= T#300ms;
            SC_OvlTesteraHV.AlarmTime.PT:= T#10s;
            SC_OvlTesteraHV.IdleTime.IN:= TRUE;

            IF SKTcpClientTester_0.Status.staReceived AND SKTcpClientTester_0.Status.DataRecv[2]= 2 AND SKTcpClientTester_0.Status.DataRecv[5]= 1 THEN
                SKTcpClientTester_0.Cmd.Send:= FALSE;
                P3_HV_Test.STAV.Vysledok_HV_Testu:= 'OK';
                SC_OvlTesteraHV.ResetStep:= TRUE;
                SC_OvlTesteraHV.Step:= 30;
            ELSIF SKTcpClientTester_0.Status.staReceived AND SKTcpClientTester_0.Status.DataRecv[2]= 2 AND SKTcpClientTester_0.Status.DataRecv[5]= 2 THEN
                SKTcpClientTester_0.Cmd.Send:= FALSE;
                P3_HV_Test.STAV.Vysledok_HV_Testu:= 'NG';
                SC_OvlTesteraHV.ResetStep:= TRUE;
                SC_OvlTesteraHV.Step:= 30;
            ELSIF SKTcpClientTester_0.Status.staReceived AND SKTcpClientTester_0.Status.DataRecv[2]= 2 AND SKTcpClientTester_0.Status.DataRecv[5]= 0 THEN
                SKTcpClientTester_0.Cmd.Send:= FALSE;
                IF SC_OvlTesteraHV.IdleTime.Q THEN
                    SC_OvlTesteraHV.ResetStep:= TRUE;
                    SC_OvlTesteraHV.Step:= 25;
                END_IF
            ELSIF SKTcpClientTester_0.Status.staReceived AND SKTcpClientTester_0.Status.DataRecv[2]= 2 AND SKTcpClientTester_0.Status.DataRecv[5]= 3 THEN
                SKTcpClientTester_0.Cmd.Send:= FALSE;
                IF SC_OvlTesteraHV.IdleTime.Q THEN
                    SC_OvlTesteraHV.ResetStep:= TRUE;
                    SC_OvlTesteraHV.Step:= 25;
                END_IF
            ELSIF SKTcpClientTester_0.Status.staError THEN
                SKTcpClientTester_0.Cmd.Send:= FALSE;
                P3_HV_Test.STAV.Vysledok_HV_Testu:= 'NG';
                P3_HV_Test.STAV.TesterNeodpoveda:= TRUE;
                SC_OvlTesteraHV.ResetStep:= TRUE;
                SC_OvlTesteraHV.Step:= 100;
            END_IF

        30:
            SC_OvlTesteraHV.StepName:= '30 - Potvrdenie precitanie vysledkov testu - typ 3';
            SC_OvlTesteraHV.IdleTime.PT:= T#300ms;
            SC_OvlTesteraHV.AlarmTime.PT:= T#10s;
            SC_OvlTesteraHV.IdleTime.IN:= TRUE;

            SKTcpClientTester_0.Params.Packet.type:= 3;
            SKTcpClientTester_0.Params.Packet.workplace:= 46;
            SKTcpClientTester_0.Params.Packet.id:= 1;
            SKTcpClientTester_0.Cmd.Send:= TRUE;

            IF SKTcpClientTester_0.Cmd.Send AND NOT SKTcpClientTester_0.Status.staReceived AND NOT SKTcpClientTester_0.Status.staError THEN
                SC_OvlTesteraHV.ResetStep:= TRUE;
                SC_OvlTesteraHV.Step:= 33;
            END_IF

        33:
            SC_OvlTesteraHV.StepName:= '33 - Odpoved testera na potvrdenie vysledkov - typ 3';
            SC_OvlTesteraHV.IdleTime.PT:= T#300ms;
            SC_OvlTesteraHV.AlarmTime.PT:= T#10s;

            IF SKTcpClientTester_0.Status.staReceived AND SKTcpClientTester_0.Status.DataRecv[2]= 3 AND SKTcpClientTester_0.Status.DataRecv[5]= 0 THEN
                SKTcpClientTester_0.Cmd.Send:= FALSE;
                P3_HV_Test.STAV.NameranyCas_CelkovyCasTestovania:= Cas_HVTester.ET;
                Cas_HVTester.IN:= FALSE;
                P3_HV_Test.STAV.TestovanieUkoncene:= TRUE;
                SC_OvlTesteraHV.ResetStep:= TRUE;
                SC_OvlTesteraHV.Step:= 100;
            ELSIF SKTcpClientTester_0.Status.staReceived AND SKTcpClientTester_0.Status.DataRecv[2]= 3 AND SKTcpClientTester_0.Status.DataRecv[5]= 1 THEN
                P3_HV_Test.STAV.Vysledok_HV_Testu:= 'NG';
                P3_HV_Test.STAV.NameranyCas_CelkovyCasTestovania:= Cas_HVTester.ET;
                Cas_HVTester.IN:= FALSE;
                P3_HV_Test.STAV.TestovanieUkoncene:= TRUE;
                SKTcpClientTester_0.Cmd.Send:= FALSE;
                SC_OvlTesteraHV.ResetStep:= TRUE;
                SC_OvlTesteraHV.Step:= 100;
            ELSIF SKTcpClientTester_0.Status.staError THEN
                SKTcpClientTester_0.Cmd.Send:= FALSE;
                P3_HV_Test.STAV.Vysledok_HV_Testu:= 'NG';
				P3_HV_Test.STAV.TesterNeodpoveda:= TRUE;
				SC_OvlTesteraHV.ResetStep:= TRUE;
                SC_OvlTesteraHV.Step:= 100;
            END_IF

        100:
            SC_OvlTesteraHV.StepName:= '100 - Cakam na zrusenie signalu start testovania';
            SC_OvlTesteraHV.IdleTime.PT:= T#3s;
            SC_OvlTesteraHV.AlarmTime.PT:= T#10s;

            IF NOT P3_HV_Test.CMD.StartTestovania THEN
                SC_OvlTesteraHV.ResetStep:= TRUE;
                SC_OvlTesteraHV.Step:= 0;
            END_IF

    END_CASE

END_ACTION
```

### Program Logical/Program/Pracovisko_3/P3_ZdvizkaPredLeakTestA (IEC)
